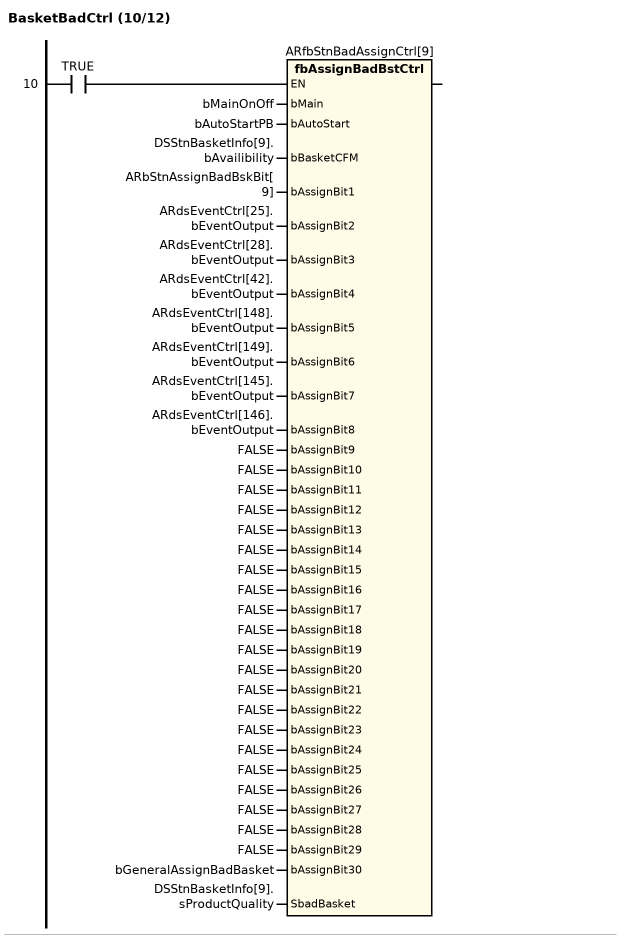
// NETWORK 10
ARfbStnBadAssignCtrl[9](
    bMain := bMainOnOff,
    bAutoStart := bAutoStartPB,
    bBasketCFM := DSStnBasketInfo[9].bAvailibility,
    bAssignBit1 := ARbStnAssignBadBskBit[9],
    bAssignBit2 := ARdsEventCtrl[25].bEventOutput,
    bAssignBit3 := ARdsEventCtrl[28].bEventOutput,
    bAssignBit4 := ARdsEventCtrl[42].bEventOutput,
    bAssignBit5 := ARdsEventCtrl[148].bEventOutput,
    bAssignBit6 := ARdsEventCtrl[149].bEventOutput,
    bAssignBit7 := ARdsEventCtrl[145].bEventOutput,
    bAssignBit8 := ARdsEventCtrl[146].bEventOutput,
    bAssignBit9 := FALSE,
    bAssignBit10 := FALSE,
    bAssignBit11 := FALSE,
    bAssignBit12 := FALSE,
    bAssignBit13 := FALSE,
    bAssignBit14 := FALSE,
    bAssignBit15 := FALSE,
    bAssignBit16 := FALSE,
    bAssignBit17 := FALSE,
    bAssignBit18 := FALSE,
    bAssignBit19 := FALSE,
    bAssignBit20 := FALSE,
    bAssignBit21 := FALSE,
    bAssignBit22 := FALSE,
    bAssignBit23 := FALSE,
    bAssignBit24 := FALSE,
    bAssignBit25 := FALSE,
    bAssignBit26 := FALSE,
    bAssignBit27 := FALSE,
    bAssignBit28 := FALSE,
    bAssignBit29 := FALSE,
    bAssignBit30 := bGeneralAssignBadBasket,
    SbadBasket := DSStnBasketInfo[9].sProductQuality); // fbAssignBadBstCtrl

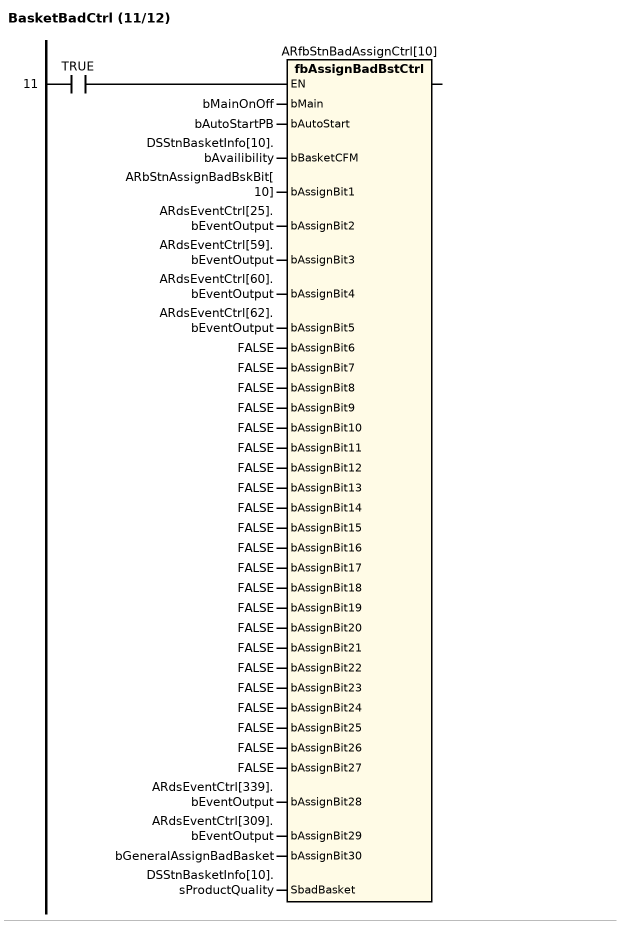
// NETWORK 11
ARfbStnBadAssignCtrl[10](
    bMain := bMainOnOff,
    bAutoStart := bAutoStartPB,
    bBasketCFM := DSStnBasketInfo[10].bAvailibility,
    bAssignBit1 := ARbStnAssignBadBskBit[10],
    bAssignBit2 := ARdsEventCtrl[25].bEventOutput,
    bAssignBit3 := ARdsEventCtrl[59].bEventOutput,
    bAssignBit4 := ARdsEventCtrl[60].bEventOutput,
    bAssignBit5 := ARdsEventCtrl[62].bEventOutput,
    bAssignBit6 := FALSE,
    bAssignBit7 := FALSE,
    bAssignBit8 := FALSE,
    bAssignBit9 := FALSE,
    bAssignBit10 := FALSE,
    bAssignBit11 := FALSE,
    bAssignBit12 := FALSE,
    bAssignBit13 := FALSE,
    bAssignBit14 := FALSE,
    bAssignBit15 := FALSE,
    bAssignBit16 := FALSE,
    bAssignBit17 := FALSE,
    bAssignBit18 := FALSE,
    bAssignBit19 := FALSE,
    bAssignBit20 := FALSE,
    bAssignBit21 := FALSE,
    bAssignBit22 := FALSE,
    bAssignBit23 := FALSE,
    bAssignBit24 := FALSE,
    bAssignBit25 := FALSE,
    bAssignBit26 := FALSE,
    bAssignBit27 := FALSE,
    bAssignBit28 := ARdsEventCtrl[339].bEventOutput,
    bAssignBit29 := ARdsEventCtrl[309].bEventOutput,
    bAssignBit30 := bGeneralAssignBadBasket,
    SbadBasket := DSStnBasketInfo[10].sProductQuality); // fbAssignBadBstCtrl

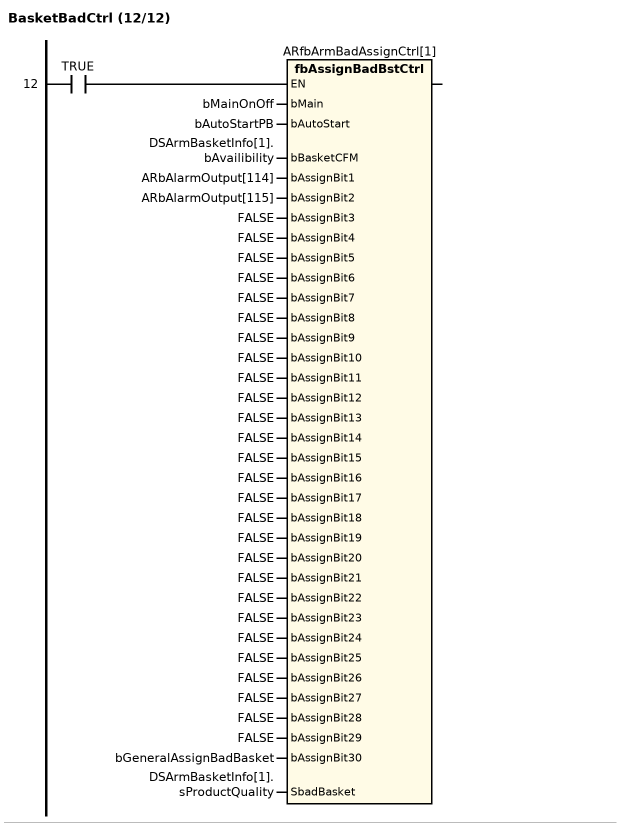
// NETWORK 12
ARfbArmBadAssignCtrl[1](
    bMain := bMainOnOff,
    bAutoStart := bAutoStartPB,
    bBasketCFM := DSArmBasketInfo[1].bAvailibility,
    bAssignBit1 := ARbAlarmOutput[114],
    bAssignBit2 := ARbAlarmOutput[115],
    bAssignBit3 := FALSE,
    bAssignBit4 := FALSE,
    bAssignBit5 := FALSE,
    bAssignBit6 := FALSE,
    bAssignBit7 := FALSE,
    bAssignBit8 := FALSE,
    bAssignBit9 := FALSE,
    bAssignBit10 := FALSE,
    bAssignBit11 := FALSE,
    bAssignBit12 := FALSE,
    bAssignBit13 := FALSE,
    bAssignBit14 := FALSE,
    bAssignBit15 := FALSE,
    bAssignBit16 := FALSE,
    bAssignBit17 := FALSE,
    bAssignBit18 := FALSE,
    bAssignBit19 := FALSE,
    bAssignBit20 := FALSE,
    bAssignBit21 := FALSE,
    bAssignBit22 := FALSE,
    bAssignBit23 := FALSE,
    bAssignBit24 := FALSE,
    bAssignBit25 := FALSE,
    bAssignBit26 := FALSE,
    bAssignBit27 := FALSE,
    bAssignBit28 := FALSE,
    bAssignBit29 := FALSE,
    bAssignBit30 := bGeneralAssignBadBasket,
    SbadBasket := DSArmBasketInfo[1].sProductQuality); // fbAssignBadBstCtrl

END_PROGRAM

// ---- FBs/B_JKS_CustomFB/fbGeneralfbFolder/fbAssignBadBstCtrl.TcPOU
FUNCTION_BLOCK fbAssignBadBstCtrl
VAR_INPUT

	bMain			: BOOL;
	bAutoStart		: BOOL;
	bBasketCFM		: BOOL;

	bAssignBit1		: BOOL;
	bAssignBit2		: BOOL;
	bAssignBit3		: BOOL;
	bAssignBit4		: BOOL;
	bAssignBit5		: BOOL;
	bAssignBit6		: BOOL;
	bAssignBit7		: BOOL;
	bAssignBit8		: BOOL;
	bAssignBit9		: BOOL;
	bAssignBit10		: BOOL;
	bAssignBit11		: BOOL;
	bAssignBit12		: BOOL;
	bAssignBit13		: BOOL;
	bAssignBit14		: BOOL;
	bAssignBit15		: BOOL;
	bAssignBit16		: BOOL;
	bAssignBit17		: BOOL;
	bAssignBit18		: BOOL;
	bAssignBit19		: BOOL;
	bAssignBit20		: BOOL;
	bAssignBit21		: BOOL;
	bAssignBit22		: BOOL;
	bAssignBit23		: BOOL;
	bAssignBit24		: BOOL;
	bAssignBit25		: BOOL;
	bAssignBit26		: BOOL;
	bAssignBit27		: BOOL;
	bAssignBit28		: BOOL;
	bAssignBit29		: BOOL;
	bAssignBit30		: BOOL;

END_VAR
VAR_IN_OUT

	SbadBasket		: STRING(50);

END_VAR
VAR
	TRIG1: R_TRIG;
END_VAR
VAR // added by the converter: edge detectors and wires of the graphical bodies
    _w1 : ANY;
END_VAR

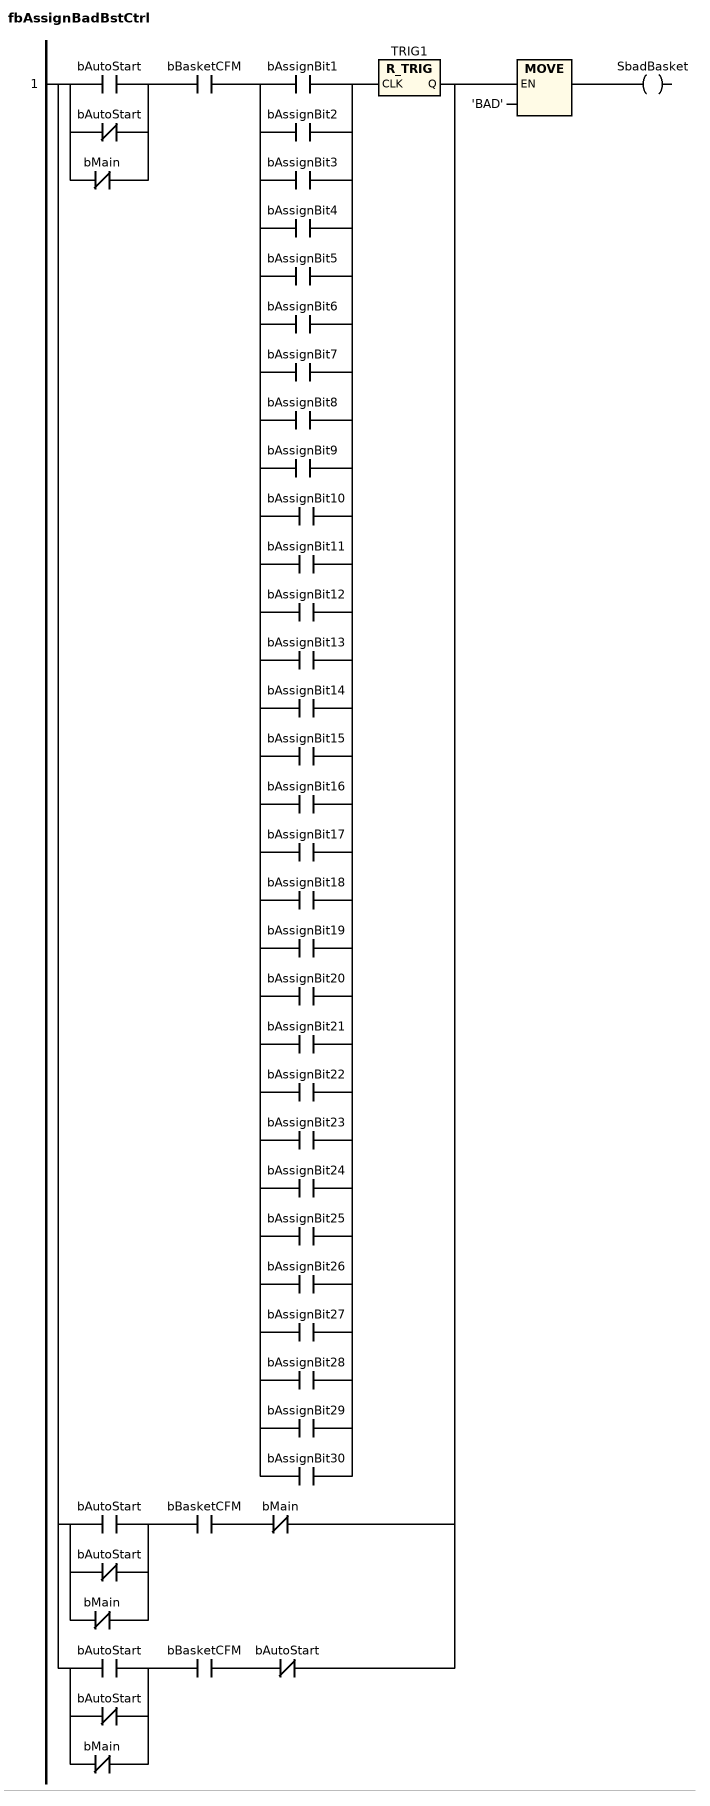
// NETWORK 1
TRIG1(CLK := ((bAutoStart OR NOT bAutoStart OR NOT bMain) AND bBasketCFM) AND (bAssignBit1 OR bAssignBit2 OR bAssignBit3 OR bAssignBit4 OR bAssignBit5 OR bAssignBit6 OR bAssignBit7 OR bAssignBit8 OR bAssignBit9 OR bAssignBit10 OR bAssignBit11 OR bAssignBit12 OR bAssignBit13 OR bAssignBit14 OR bAssignBit15 OR bAssignBit16 OR bAssignBit17 OR bAssignBit18 OR bAssignBit19 OR bAssignBit20 OR bAssignBit21 OR bAssignBit22 OR bAssignBit23 OR bAssignBit24 OR bAssignBit25 OR bAssignBit26 OR bAssignBit27 OR bAssignBit28 OR bAssignBit29 OR bAssignBit30)); // R_TRIG
IF TRIG1.Q OR ((bAutoStart OR NOT bAutoStart OR NOT bMain) AND bBasketCFM) AND NOT bMain OR ((bAutoStart OR NOT bAutoStart OR NOT bMain) AND bBasketCFM) AND NOT bAutoStart THEN
    _w1 := 'BAD';
END_IF
SbadBasket := _w1;

END_FUNCTION_BLOCK

// ---- POUs/MainProgram/BasketMemory_RecipeCtrl/BasketMemoryCtrl.TcPOU
PROGRAM BasketMemoryCtrl
VAR

	NIL: BOOL;

END_VAR

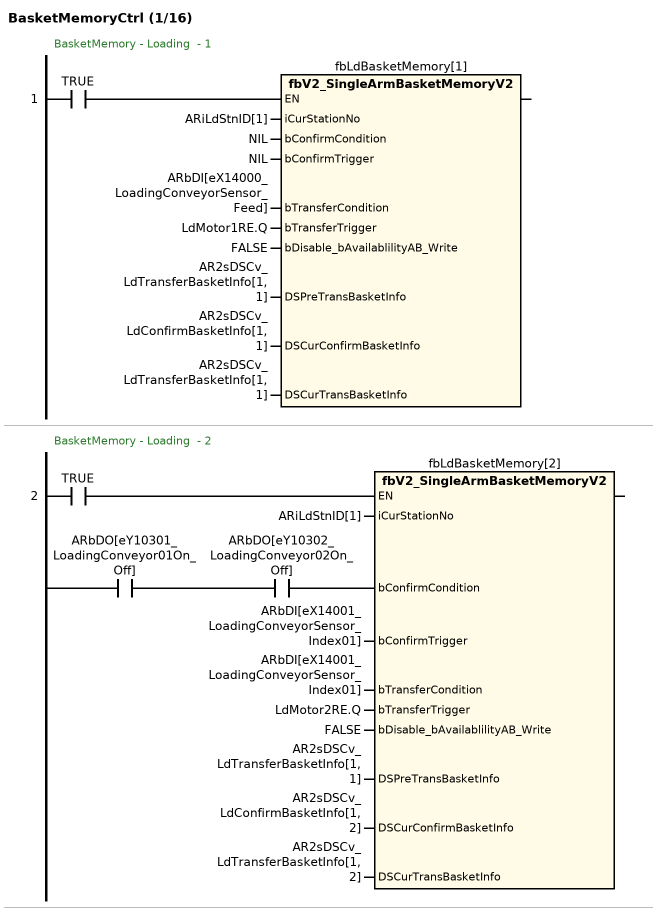
// NETWORK 1
// BasketMemory - Loading  - 1
fbLdBasketMemory[1](
    iCurStationNo := ARiLdStnID[1],
    bConfirmCondition := NIL,
    bConfirmTrigger := NIL,
    bTransferCondition := ARbDI[eX14000_LoadingConveyorSensor_Feed],
    bTransferTrigger := LdMotor1RE.Q,
    bDisable_bAvailablilityAB_Write := FALSE,
    DSPreTransBasketInfo := AR2sDSCv_LdTransferBasketInfo[1,1],
    DSCurConfirmBasketInfo := AR2sDSCv_LdConfirmBasketInfo[1,1],
    DSCurTransBasketInfo := AR2sDSCv_LdTransferBasketInfo[1,1]); // fbV2_SingleArmBasketMemoryV2

// NETWORK 2
// BasketMemory - Loading  - 2
fbLdBasketMemory[2](
    iCurStationNo := ARiLdStnID[1],
    bConfirmCondition := ARbDO[eY10301_LoadingConveyor01On_Off] AND ARbDO[eY10302_LoadingConveyor02On_Off],
    bConfirmTrigger := ARbDI[eX14001_LoadingConveyorSensor_Index01],
    bTransferCondition := ARbDI[eX14001_LoadingConveyorSensor_Index01],
    bTransferTrigger := LdMotor2RE.Q,
    bDisable_bAvailablilityAB_Write := FALSE,
    DSPreTransBasketInfo := AR2sDSCv_LdTransferBasketInfo[1,1],
    DSCurConfirmBasketInfo := AR2sDSCv_LdConfirmBasketInfo[1,2],
    DSCurTransBasketInfo := AR2sDSCv_LdTransferBasketInfo[1,2]); // fbV2_SingleArmBasketMemoryV2

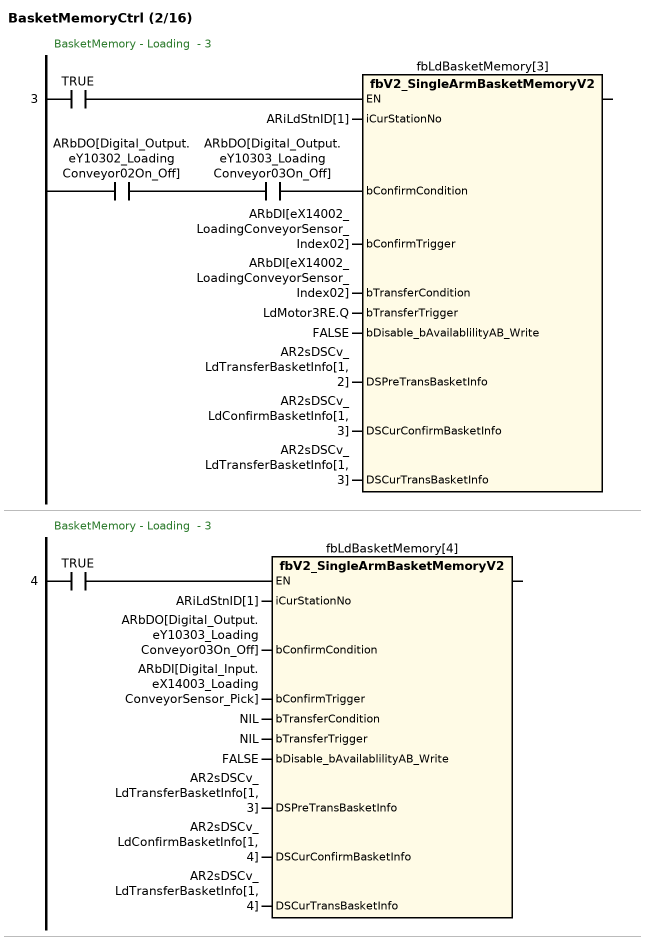
// NETWORK 3
// BasketMemory - Loading  - 3
fbLdBasketMemory[3](
    iCurStationNo := ARiLdStnID[1],
    bConfirmCondition := ARbDO[Digital_Output.eY10302_LoadingConveyor02On_Off] AND ARbDO[Digital_Output.eY10303_LoadingConveyor03On_Off],
    bConfirmTrigger := ARbDI[eX14002_LoadingConveyorSensor_Index02],
    bTransferCondition := ARbDI[eX14002_LoadingConveyorSensor_Index02],
    bTransferTrigger := LdMotor3RE.Q,
    bDisable_bAvailablilityAB_Write := FALSE,
    DSPreTransBasketInfo := AR2sDSCv_LdTransferBasketInfo[1,2],
    DSCurConfirmBasketInfo := AR2sDSCv_LdConfirmBasketInfo[1,3],
    DSCurTransBasketInfo := AR2sDSCv_LdTransferBasketInfo[1,3]); // fbV2_SingleArmBasketMemoryV2

// NETWORK 4
// BasketMemory - Loading  - 3
fbLdBasketMemory[4](
    iCurStationNo := ARiLdStnID[1],
    bConfirmCondition := ARbDO[Digital_Output.eY10303_LoadingConveyor03On_Off],
    bConfirmTrigger := ARbDI[Digital_Input.eX14003_LoadingConveyorSensor_Pick],
    bTransferCondition := NIL,
    bTransferTrigger := NIL,
    bDisable_bAvailablilityAB_Write := FALSE,
    DSPreTransBasketInfo := AR2sDSCv_LdTransferBasketInfo[1,3],
    DSCurConfirmBasketInfo := AR2sDSCv_LdConfirmBasketInfo[1,4],
    DSCurTransBasketInfo := AR2sDSCv_LdTransferBasketInfo[1,4]); // fbV2_SingleArmBasketMemoryV2

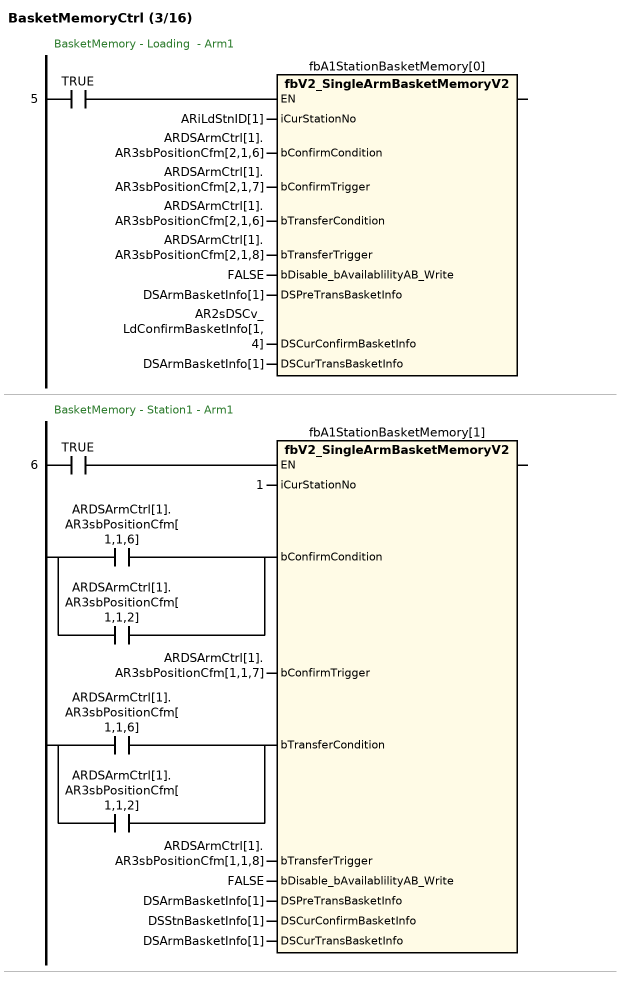
// NETWORK 5
// BasketMemory - Loading  - Arm1
fbA1StationBasketMemory[0](
    iCurStationNo := ARiLdStnID[1],
    bConfirmCondition := ARDSArmCtrl[1].AR3sbPositionCfm[2,1,6],
    bConfirmTrigger := ARDSArmCtrl[1].AR3sbPositionCfm[2,1,7],
    bTransferCondition := ARDSArmCtrl[1].AR3sbPositionCfm[2,1,6],
    bTransferTrigger := ARDSArmCtrl[1].AR3sbPositionCfm[2,1,8],
    bDisable_bAvailablilityAB_Write := FALSE,
    DSPreTransBasketInfo := DSArmBasketInfo[1],
    DSCurConfirmBasketInfo := AR2sDSCv_LdConfirmBasketInfo[1,4],
    DSCurTransBasketInfo := DSArmBasketInfo[1]); // fbV2_SingleArmBasketMemoryV2

// NETWORK 6
// BasketMemory - Station1 - Arm1
fbA1StationBasketMemory[1](
    iCurStationNo := 1,
    bConfirmCondition := ARDSArmCtrl[1].AR3sbPositionCfm[1,1,6] OR ARDSArmCtrl[1].AR3sbPositionCfm[1,1,2],
    bConfirmTrigger := ARDSArmCtrl[1].AR3sbPositionCfm[1,1,7],
    bTransferCondition := ARDSArmCtrl[1].AR3sbPositionCfm[1,1,6] OR ARDSArmCtrl[1].AR3sbPositionCfm[1,1,2],
    bTransferTrigger := ARDSArmCtrl[1].AR3sbPositionCfm[1,1,8],
    bDisable_bAvailablilityAB_Write := FALSE,
    DSPreTransBasketInfo := DSArmBasketInfo[1],
    DSCurConfirmBasketInfo := DSStnBasketInfo[1],
    DSCurTransBasketInfo := DSArmBasketInfo[1]); // fbV2_SingleArmBasketMemoryV2

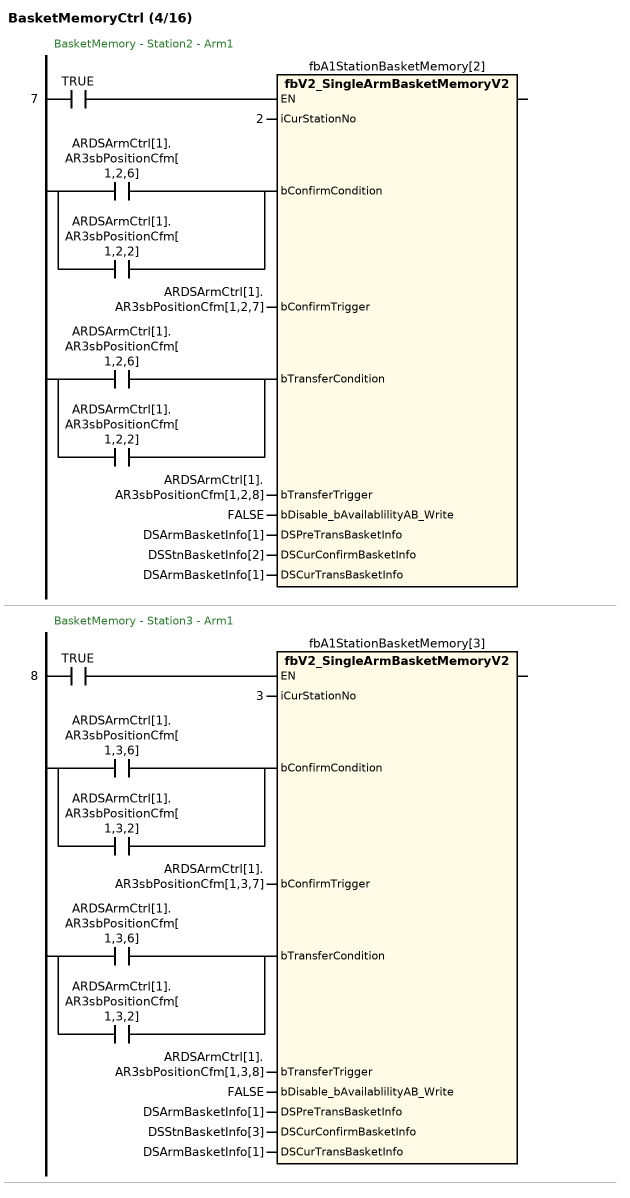
// NETWORK 7
// BasketMemory - Station2 - Arm1
fbA1StationBasketMemory[2](
    iCurStationNo := 2,
    bConfirmCondition := ARDSArmCtrl[1].AR3sbPositionCfm[1,2,6] OR ARDSArmCtrl[1].AR3sbPositionCfm[1,2,2],
    bConfirmTrigger := ARDSArmCtrl[1].AR3sbPositionCfm[1,2,7],
    bTransferCondition := ARDSArmCtrl[1].AR3sbPositionCfm[1,2,6] OR ARDSArmCtrl[1].AR3sbPositionCfm[1,2,2],
    bTransferTrigger := ARDSArmCtrl[1].AR3sbPositionCfm[1,2,8],
    bDisable_bAvailablilityAB_Write := FALSE,
    DSPreTransBasketInfo := DSArmBasketInfo[1],
    DSCurConfirmBasketInfo := DSStnBasketInfo[2],
    DSCurTransBasketInfo := DSArmBasketInfo[1]); // fbV2_SingleArmBasketMemoryV2

// NETWORK 8
// BasketMemory - Station3 - Arm1
fbA1StationBasketMemory[3](
    iCurStationNo := 3,
    bConfirmCondition := ARDSArmCtrl[1].AR3sbPositionCfm[1,3,6] OR ARDSArmCtrl[1].AR3sbPositionCfm[1,3,2],
    bConfirmTrigger := ARDSArmCtrl[1].AR3sbPositionCfm[1,3,7],
    bTransferCondition := ARDSArmCtrl[1].AR3sbPositionCfm[1,3,6] OR ARDSArmCtrl[1].AR3sbPositionCfm[1,3,2],
    bTransferTrigger := ARDSArmCtrl[1].AR3sbPositionCfm[1,3,8],
    bDisable_bAvailablilityAB_Write := FALSE,
    DSPreTransBasketInfo := DSArmBasketInfo[1],
    DSCurConfirmBasketInfo := DSStnBasketInfo[3],
    DSCurTransBasketInfo := DSArmBasketInfo[1]); // fbV2_SingleArmBasketMemoryV2

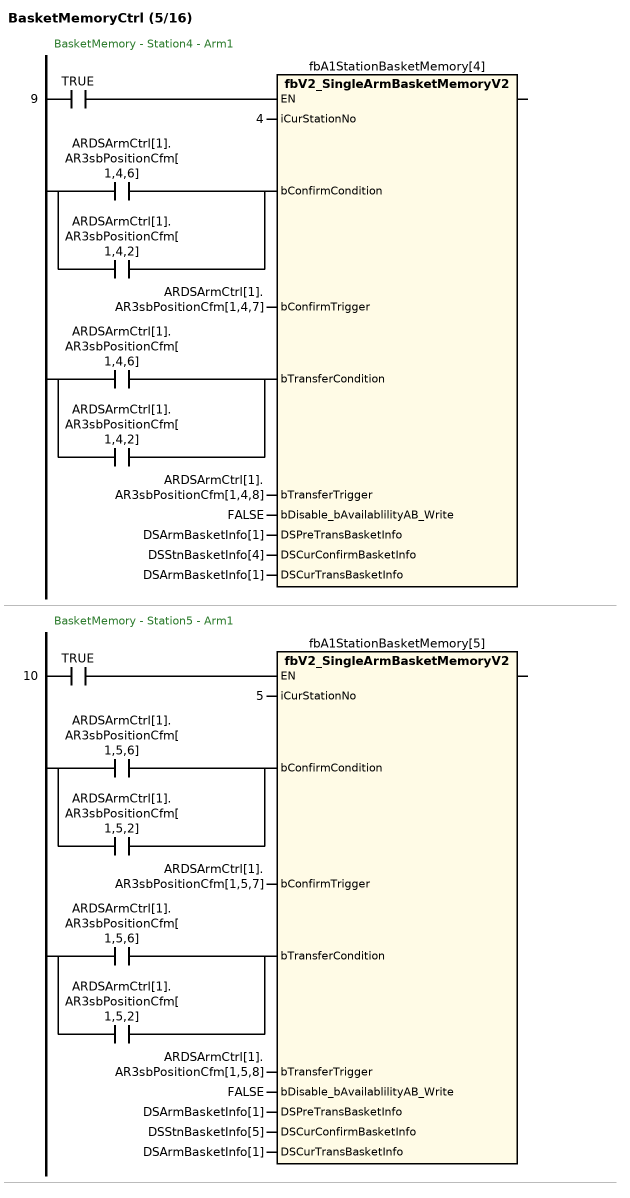
// NETWORK 9
// BasketMemory - Station4 - Arm1
fbA1StationBasketMemory[4](
    iCurStationNo := 4,
    bConfirmCondition := ARDSArmCtrl[1].AR3sbPositionCfm[1,4,6] OR ARDSArmCtrl[1].AR3sbPositionCfm[1,4,2],
    bConfirmTrigger := ARDSArmCtrl[1].AR3sbPositionCfm[1,4,7],
    bTransferCondition := ARDSArmCtrl[1].AR3sbPositionCfm[1,4,6] OR ARDSArmCtrl[1].AR3sbPositionCfm[1,4,2],
    bTransferTrigger := ARDSArmCtrl[1].AR3sbPositionCfm[1,4,8],
    bDisable_bAvailablilityAB_Write := FALSE,
    DSPreTransBasketInfo := DSArmBasketInfo[1],
    DSCurConfirmBasketInfo := DSStnBasketInfo[4],
    DSCurTransBasketInfo := DSArmBasketInfo[1]); // fbV2_SingleArmBasketMemoryV2

// NETWORK 10
// BasketMemory - Station5 - Arm1
fbA1StationBasketMemory[5](
    iCurStationNo := 5,
    bConfirmCondition := ARDSArmCtrl[1].AR3sbPositionCfm[1,5,6] OR ARDSArmCtrl[1].AR3sbPositionCfm[1,5,2],
    bConfirmTrigger := ARDSArmCtrl[1].AR3sbPositionCfm[1,5,7],
    bTransferCondition := ARDSArmCtrl[1].AR3sbPositionCfm[1,5,6] OR ARDSArmCtrl[1].AR3sbPositionCfm[1,5,2],
    bTransferTrigger := ARDSArmCtrl[1].AR3sbPositionCfm[1,5,8],
    bDisable_bAvailablilityAB_Write := FALSE,
    DSPreTransBasketInfo := DSArmBasketInfo[1],
    DSCurConfirmBasketInfo := DSStnBasketInfo[5],
    DSCurTransBasketInfo := DSArmBasketInfo[1]); // fbV2_SingleArmBasketMemoryV2

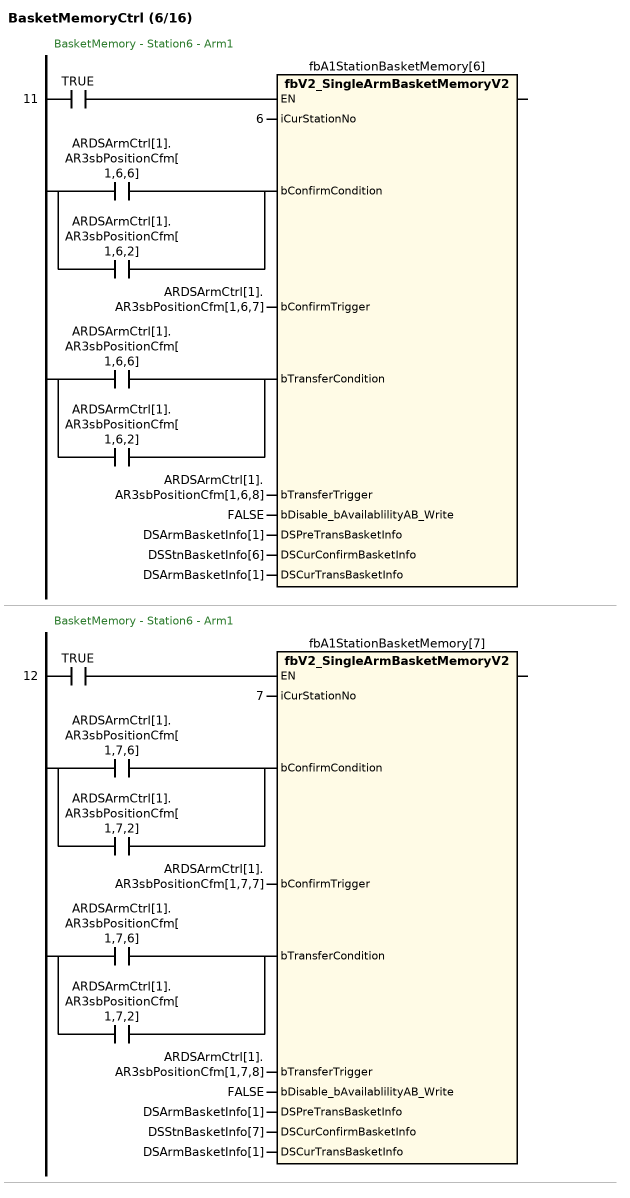
// NETWORK 11
// BasketMemory - Station6 - Arm1
fbA1StationBasketMemory[6](
    iCurStationNo := 6,
    bConfirmCondition := ARDSArmCtrl[1].AR3sbPositionCfm[1,6,6] OR ARDSArmCtrl[1].AR3sbPositionCfm[1,6,2],
    bConfirmTrigger := ARDSArmCtrl[1].AR3sbPositionCfm[1,6,7],
    bTransferCondition := ARDSArmCtrl[1].AR3sbPositionCfm[1,6,6] OR ARDSArmCtrl[1].AR3sbPositionCfm[1,6,2],
    bTransferTrigger := ARDSArmCtrl[1].AR3sbPositionCfm[1,6,8],
    bDisable_bAvailablilityAB_Write := FALSE,
    DSPreTransBasketInfo := DSArmBasketInfo[1],
    DSCurConfirmBasketInfo := DSStnBasketInfo[6],
    DSCurTransBasketInfo := DSArmBasketInfo[1]); // fbV2_SingleArmBasketMemoryV2

// NETWORK 12
// BasketMemory - Station6 - Arm1
fbA1StationBasketMemory[7](
    iCurStationNo := 7,
    bConfirmCondition := ARDSArmCtrl[1].AR3sbPositionCfm[1,7,6] OR ARDSArmCtrl[1].AR3sbPositionCfm[1,7,2],
    bConfirmTrigger := ARDSArmCtrl[1].AR3sbPositionCfm[1,7,7],
    bTransferCondition := ARDSArmCtrl[1].AR3sbPositionCfm[1,7,6] OR ARDSArmCtrl[1].AR3sbPositionCfm[1,7,2],
    bTransferTrigger := ARDSArmCtrl[1].AR3sbPositionCfm[1,7,8],
    bDisable_bAvailablilityAB_Write := FALSE,
    DSPreTransBasketInfo := DSArmBasketInfo[1],
    DSCurConfirmBasketInfo := DSStnBasketInfo[7],
    DSCurTransBasketInfo := DSArmBasketInfo[1]); // fbV2_SingleArmBasketMemoryV2

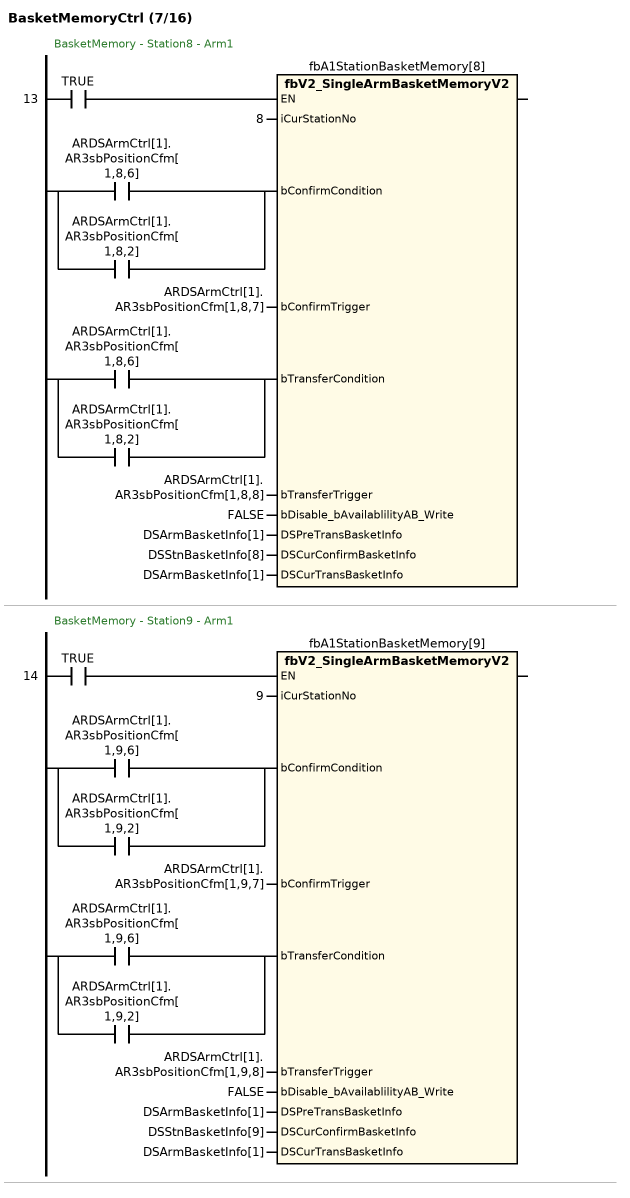
// NETWORK 13
// BasketMemory - Station8 - Arm1
fbA1StationBasketMemory[8](
    iCurStationNo := 8,
    bConfirmCondition := ARDSArmCtrl[1].AR3sbPositionCfm[1,8,6] OR ARDSArmCtrl[1].AR3sbPositionCfm[1,8,2],
    bConfirmTrigger := ARDSArmCtrl[1].AR3sbPositionCfm[1,8,7],
    bTransferCondition := ARDSArmCtrl[1].AR3sbPositionCfm[1,8,6] OR ARDSArmCtrl[1].AR3sbPositionCfm[1,8,2],
    bTransferTrigger := ARDSArmCtrl[1].AR3sbPositionCfm[1,8,8],
    bDisable_bAvailablilityAB_Write := FALSE,
    DSPreTransBasketInfo := DSArmBasketInfo[1],
    DSCurConfirmBasketInfo := DSStnBasketInfo[8],
    DSCurTransBasketInfo := DSArmBasketInfo[1]); // fbV2_SingleArmBasketMemoryV2

// NETWORK 14
// BasketMemory - Station9 - Arm1
fbA1StationBasketMemory[9](
    iCurStationNo := 9,
    bConfirmCondition := ARDSArmCtrl[1].AR3sbPositionCfm[1,9,6] OR ARDSArmCtrl[1].AR3sbPositionCfm[1,9,2],
    bConfirmTrigger := ARDSArmCtrl[1].AR3sbPositionCfm[1,9,7],
    bTransferCondition := ARDSArmCtrl[1].AR3sbPositionCfm[1,9,6] OR ARDSArmCtrl[1].AR3sbPositionCfm[1,9,2],
    bTransferTrigger := ARDSArmCtrl[1].AR3sbPositionCfm[1,9,8],
    bDisable_bAvailablilityAB_Write := FALSE,
    DSPreTransBasketInfo := DSArmBasketInfo[1],
    DSCurConfirmBasketInfo := DSStnBasketInfo[9],
    DSCurTransBasketInfo := DSArmBasketInfo[1]); // fbV2_SingleArmBasketMemoryV2

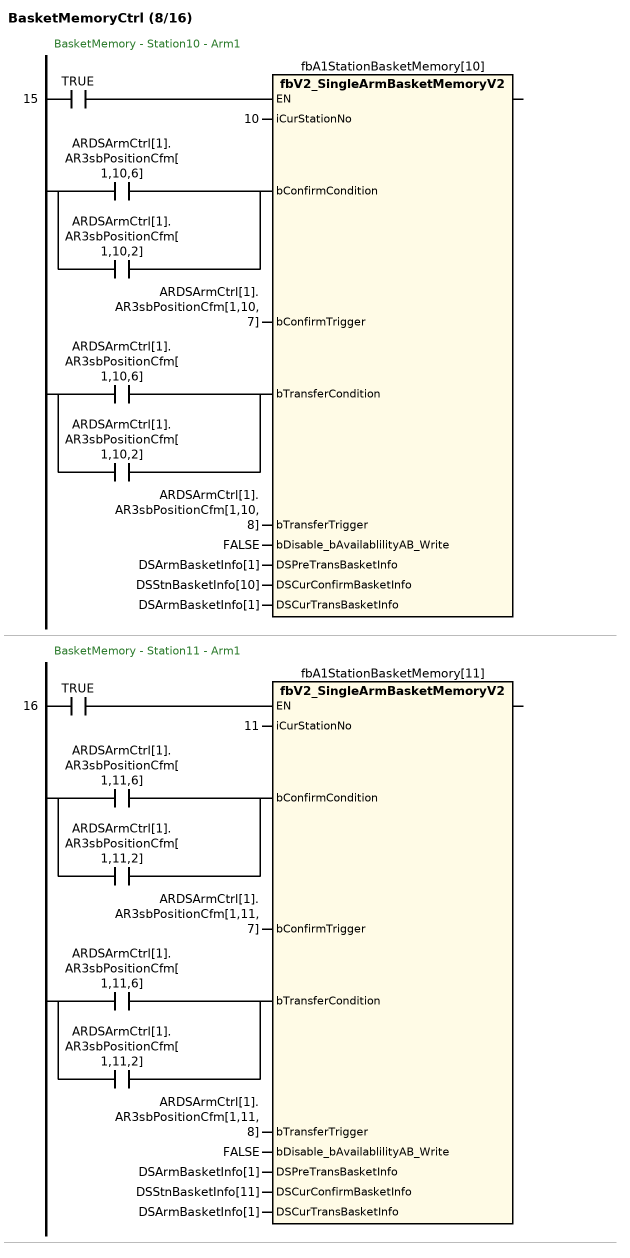
// NETWORK 15
// BasketMemory - Station10 - Arm1
fbA1StationBasketMemory[10](
    iCurStationNo := 10,
    bConfirmCondition := ARDSArmCtrl[1].AR3sbPositionCfm[1,10,6] OR ARDSArmCtrl[1].AR3sbPositionCfm[1,10,2],
    bConfirmTrigger := ARDSArmCtrl[1].AR3sbPositionCfm[1,10,7],
    bTransferCondition := ARDSArmCtrl[1].AR3sbPositionCfm[1,10,6] OR ARDSArmCtrl[1].AR3sbPositionCfm[1,10,2],
    bTransferTrigger := ARDSArmCtrl[1].AR3sbPositionCfm[1,10,8],
    bDisable_bAvailablilityAB_Write := FALSE,
    DSPreTransBasketInfo := DSArmBasketInfo[1],
    DSCurConfirmBasketInfo := DSStnBasketInfo[10],
    DSCurTransBasketInfo := DSArmBasketInfo[1]); // fbV2_SingleArmBasketMemoryV2

// NETWORK 16
// BasketMemory - Station11 - Arm1
fbA1StationBasketMemory[11](
    iCurStationNo := 11,
    bConfirmCondition := ARDSArmCtrl[1].AR3sbPositionCfm[1,11,6] OR ARDSArmCtrl[1].AR3sbPositionCfm[1,11,2],
    bConfirmTrigger := ARDSArmCtrl[1].AR3sbPositionCfm[1,11,7],
    bTransferCondition := ARDSArmCtrl[1].AR3sbPositionCfm[1,11,6] OR ARDSArmCtrl[1].AR3sbPositionCfm[1,11,2],
    bTransferTrigger := ARDSArmCtrl[1].AR3sbPositionCfm[1,11,8],
    bDisable_bAvailablilityAB_Write := FALSE,
    DSPreTransBasketInfo := DSArmBasketInfo[1],
    DSCurConfirmBasketInfo := DSStnBasketInfo[11],
    DSCurTransBasketInfo := DSArmBasketInfo[1]); // fbV2_SingleArmBasketMemoryV2

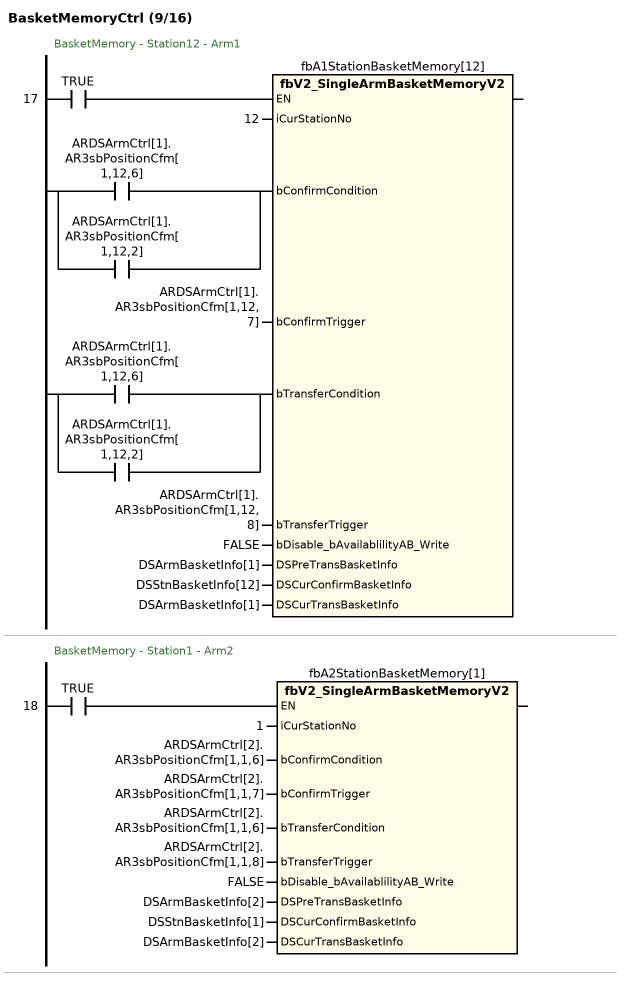
// NETWORK 17
// BasketMemory - Station12 - Arm1
fbA1StationBasketMemory[12](
    iCurStationNo := 12,
    bConfirmCondition := ARDSArmCtrl[1].AR3sbPositionCfm[1,12,6] OR ARDSArmCtrl[1].AR3sbPositionCfm[1,12,2],
    bConfirmTrigger := ARDSArmCtrl[1].AR3sbPositionCfm[1,12,7],
    bTransferCondition := ARDSArmCtrl[1].AR3sbPositionCfm[1,12,6] OR ARDSArmCtrl[1].AR3sbPositionCfm[1,12,2],
    bTransferTrigger := ARDSArmCtrl[1].AR3sbPositionCfm[1,12,8],
    bDisable_bAvailablilityAB_Write := FALSE,
    DSPreTransBasketInfo := DSArmBasketInfo[1],
    DSCurConfirmBasketInfo := DSStnBasketInfo[12],
    DSCurTransBasketInfo := DSArmBasketInfo[1]); // fbV2_SingleArmBasketMemoryV2

// NETWORK 18
// BasketMemory - Station1 - Arm2
fbA2StationBasketMemory[1](
    iCurStationNo := 1,
    bConfirmCondition := ARDSArmCtrl[2].AR3sbPositionCfm[1,1,6],
    bConfirmTrigger := ARDSArmCtrl[2].AR3sbPositionCfm[1,1,7],
    bTransferCondition := ARDSArmCtrl[2].AR3sbPositionCfm[1,1,6],
    bTransferTrigger := ARDSArmCtrl[2].AR3sbPositionCfm[1,1,8],
    bDisable_bAvailablilityAB_Write := FALSE,
    DSPreTransBasketInfo := DSArmBasketInfo[2],
    DSCurConfirmBasketInfo := DSStnBasketInfo[1],
    DSCurTransBasketInfo := DSArmBasketInfo[2]); // fbV2_SingleArmBasketMemoryV2

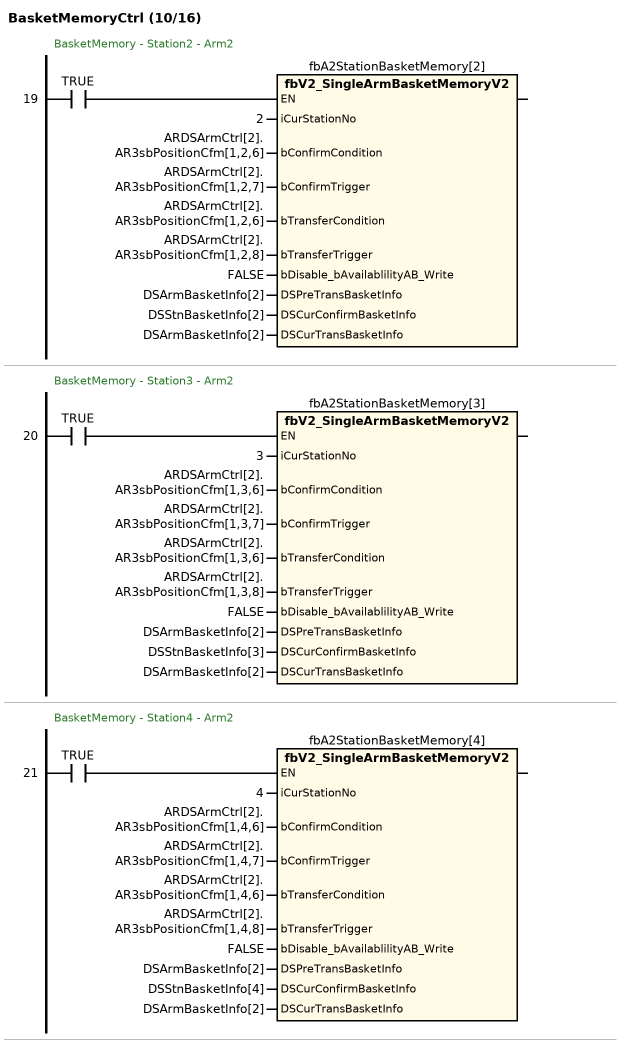
// NETWORK 19
// BasketMemory - Station2 - Arm2
fbA2StationBasketMemory[2](
    iCurStationNo := 2,
    bConfirmCondition := ARDSArmCtrl[2].AR3sbPositionCfm[1,2,6],
    bConfirmTrigger := ARDSArmCtrl[2].AR3sbPositionCfm[1,2,7],
    bTransferCondition := ARDSArmCtrl[2].AR3sbPositionCfm[1,2,6],
    bTransferTrigger := ARDSArmCtrl[2].AR3sbPositionCfm[1,2,8],
    bDisable_bAvailablilityAB_Write := FALSE,
    DSPreTransBasketInfo := DSArmBasketInfo[2],
    DSCurConfirmBasketInfo := DSStnBasketInfo[2],
    DSCurTransBasketInfo := DSArmBasketInfo[2]); // fbV2_SingleArmBasketMemoryV2

// NETWORK 20
// BasketMemory - Station3 - Arm2
fbA2StationBasketMemory[3](
    iCurStationNo := 3,
    bConfirmCondition := ARDSArmCtrl[2].AR3sbPositionCfm[1,3,6],
    bConfirmTrigger := ARDSArmCtrl[2].AR3sbPositionCfm[1,3,7],
    bTransferCondition := ARDSArmCtrl[2].AR3sbPositionCfm[1,3,6],
    bTransferTrigger := ARDSArmCtrl[2].AR3sbPositionCfm[1,3,8],
    bDisable_bAvailablilityAB_Write := FALSE,
    DSPreTransBasketInfo := DSArmBasketInfo[2],
    DSCurConfirmBasketInfo := DSStnBasketInfo[3],
    DSCurTransBasketInfo := DSArmBasketInfo[2]); // fbV2_SingleArmBasketMemoryV2

// NETWORK 21
// BasketMemory - Station4 - Arm2
fbA2StationBasketMemory[4](
    iCurStationNo := 4,
    bConfirmCondition := ARDSArmCtrl[2].AR3sbPositionCfm[1,4,6],
    bConfirmTrigger := ARDSArmCtrl[2].AR3sbPositionCfm[1,4,7],
    bTransferCondition := ARDSArmCtrl[2].AR3sbPositionCfm[1,4,6],
    bTransferTrigger := ARDSArmCtrl[2].AR3sbPositionCfm[1,4,8],
    bDisable_bAvailablilityAB_Write := FALSE,
    DSPreTransBasketInfo := DSArmBasketInfo[2],
    DSCurConfirmBasketInfo := DSStnBasketInfo[4],
    DSCurTransBasketInfo := DSArmBasketInfo[2]); // fbV2_SingleArmBasketMemoryV2

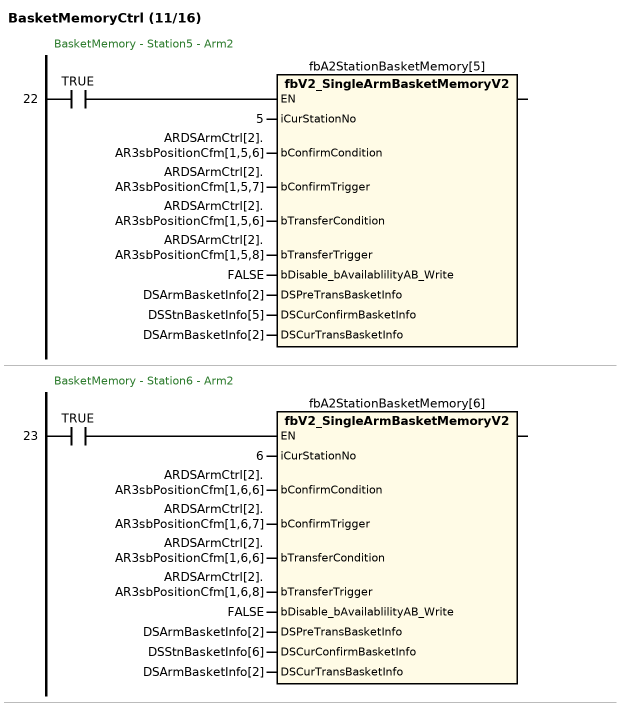
// NETWORK 22
// BasketMemory - Station5 - Arm2
fbA2StationBasketMemory[5](
    iCurStationNo := 5,
    bConfirmCondition := ARDSArmCtrl[2].AR3sbPositionCfm[1,5,6],
    bConfirmTrigger := ARDSArmCtrl[2].AR3sbPositionCfm[1,5,7],
    bTransferCondition := ARDSArmCtrl[2].AR3sbPositionCfm[1,5,6],
    bTransferTrigger := ARDSArmCtrl[2].AR3sbPositionCfm[1,5,8],
    bDisable_bAvailablilityAB_Write := FALSE,
    DSPreTransBasketInfo := DSArmBasketInfo[2],
    DSCurConfirmBasketInfo := DSStnBasketInfo[5],
    DSCurTransBasketInfo := DSArmBasketInfo[2]); // fbV2_SingleArmBasketMemoryV2

// NETWORK 23
// BasketMemory - Station6 - Arm2
fbA2StationBasketMemory[6](
    iCurStationNo := 6,
    bConfirmCondition := ARDSArmCtrl[2].AR3sbPositionCfm[1,6,6],
    bConfirmTrigger := ARDSArmCtrl[2].AR3sbPositionCfm[1,6,7],
    bTransferCondition := ARDSArmCtrl[2].AR3sbPositionCfm[1,6,6],
    bTransferTrigger := ARDSArmCtrl[2].AR3sbPositionCfm[1,6,8],
    bDisable_bAvailablilityAB_Write := FALSE,
    DSPreTransBasketInfo := DSArmBasketInfo[2],
    DSCurConfirmBasketInfo := DSStnBasketInfo[6],
    DSCurTransBasketInfo := DSArmBasketInfo[2]); // fbV2_SingleArmBasketMemoryV2

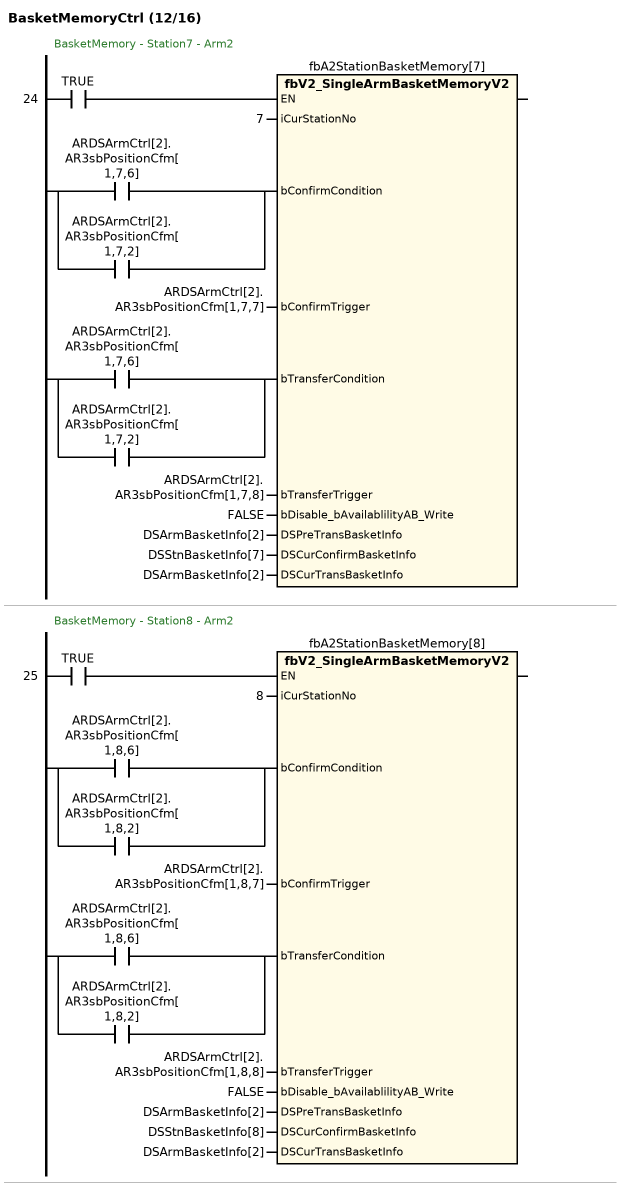
// NETWORK 24
// BasketMemory - Station7 - Arm2
fbA2StationBasketMemory[7](
    iCurStationNo := 7,
    bConfirmCondition := ARDSArmCtrl[2].AR3sbPositionCfm[1,7,6] OR ARDSArmCtrl[2].AR3sbPositionCfm[1,7,2],
    bConfirmTrigger := ARDSArmCtrl[2].AR3sbPositionCfm[1,7,7],
    bTransferCondition := ARDSArmCtrl[2].AR3sbPositionCfm[1,7,6] OR ARDSArmCtrl[2].AR3sbPositionCfm[1,7,2],
    bTransferTrigger := ARDSArmCtrl[2].AR3sbPositionCfm[1,7,8],
    bDisable_bAvailablilityAB_Write := FALSE,
    DSPreTransBasketInfo := DSArmBasketInfo[2],
    DSCurConfirmBasketInfo := DSStnBasketInfo[7],
    DSCurTransBasketInfo := DSArmBasketInfo[2]); // fbV2_SingleArmBasketMemoryV2

// NETWORK 25
// BasketMemory - Station8 - Arm2
fbA2StationBasketMemory[8](
    iCurStationNo := 8,
    bConfirmCondition := ARDSArmCtrl[2].AR3sbPositionCfm[1,8,6] OR ARDSArmCtrl[2].AR3sbPositionCfm[1,8,2],
    bConfirmTrigger := ARDSArmCtrl[2].AR3sbPositionCfm[1,8,7],
    bTransferCondition := ARDSArmCtrl[2].AR3sbPositionCfm[1,8,6] OR ARDSArmCtrl[2].AR3sbPositionCfm[1,8,2],
    bTransferTrigger := ARDSArmCtrl[2].AR3sbPositionCfm[1,8,8],
    bDisable_bAvailablilityAB_Write := FALSE,
    DSPreTransBasketInfo := DSArmBasketInfo[2],
    DSCurConfirmBasketInfo := DSStnBasketInfo[8],
    DSCurTransBasketInfo := DSArmBasketInfo[2]); // fbV2_SingleArmBasketMemoryV2

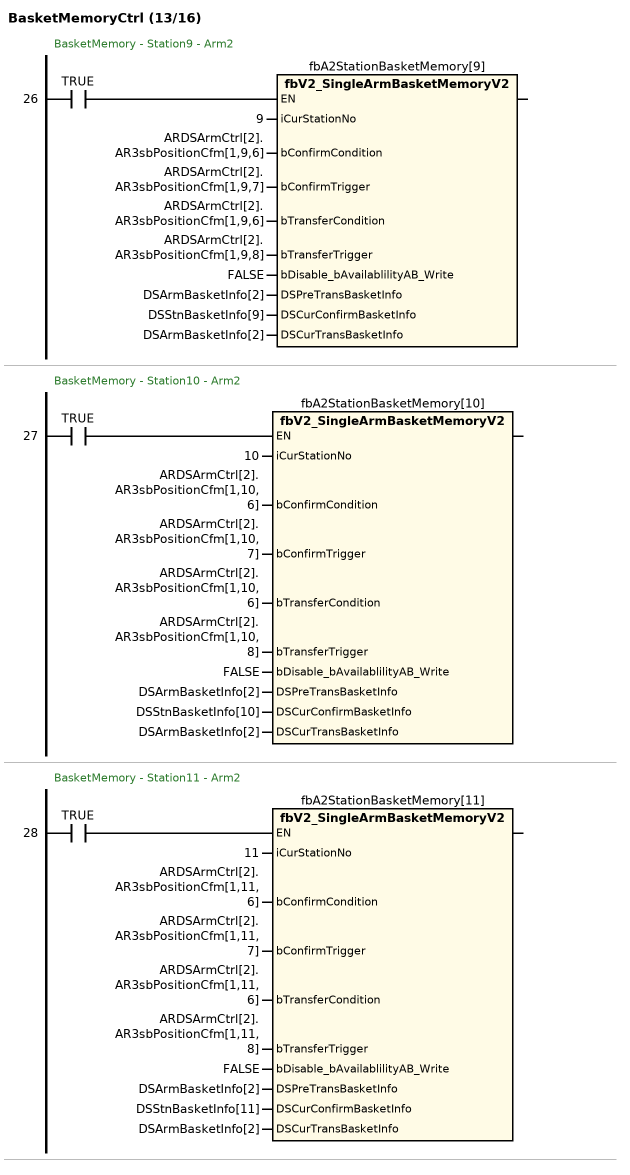
// NETWORK 26
// BasketMemory - Station9 - Arm2
fbA2StationBasketMemory[9](
    iCurStationNo := 9,
    bConfirmCondition := ARDSArmCtrl[2].AR3sbPositionCfm[1,9,6],
    bConfirmTrigger := ARDSArmCtrl[2].AR3sbPositionCfm[1,9,7],
    bTransferCondition := ARDSArmCtrl[2].AR3sbPositionCfm[1,9,6],
    bTransferTrigger := ARDSArmCtrl[2].AR3sbPositionCfm[1,9,8],
    bDisable_bAvailablilityAB_Write := FALSE,
    DSPreTransBasketInfo := DSArmBasketInfo[2],
    DSCurConfirmBasketInfo := DSStnBasketInfo[9],
    DSCurTransBasketInfo := DSArmBasketInfo[2]); // fbV2_SingleArmBasketMemoryV2

// NETWORK 27
// BasketMemory - Station10 - Arm2
fbA2StationBasketMemory[10](
    iCurStationNo := 10,
    bConfirmCondition := ARDSArmCtrl[2].AR3sbPositionCfm[1,10,6],
    bConfirmTrigger := ARDSArmCtrl[2].AR3sbPositionCfm[1,10,7],
    bTransferCondition := ARDSArmCtrl[2].AR3sbPositionCfm[1,10,6],
    bTransferTrigger := ARDSArmCtrl[2].AR3sbPositionCfm[1,10,8],
    bDisable_bAvailablilityAB_Write := FALSE,
    DSPreTransBasketInfo := DSArmBasketInfo[2],
    DSCurConfirmBasketInfo := DSStnBasketInfo[10],
    DSCurTransBasketInfo := DSArmBasketInfo[2]); // fbV2_SingleArmBasketMemoryV2

// NETWORK 28
// BasketMemory - Station11 - Arm2
fbA2StationBasketMemory[11](
    iCurStationNo := 11,
    bConfirmCondition := ARDSArmCtrl[2].AR3sbPositionCfm[1,11,6],
    bConfirmTrigger := ARDSArmCtrl[2].AR3sbPositionCfm[1,11,7],
    bTransferCondition := ARDSArmCtrl[2].AR3sbPositionCfm[1,11,6],
    bTransferTrigger := ARDSArmCtrl[2].AR3sbPositionCfm[1,11,8],
    bDisable_bAvailablilityAB_Write := FALSE,
    DSPreTransBasketInfo := DSArmBasketInfo[2],
    DSCurConfirmBasketInfo := DSStnBasketInfo[11],
    DSCurTransBasketInfo := DSArmBasketInfo[2]); // fbV2_SingleArmBasketMemoryV2

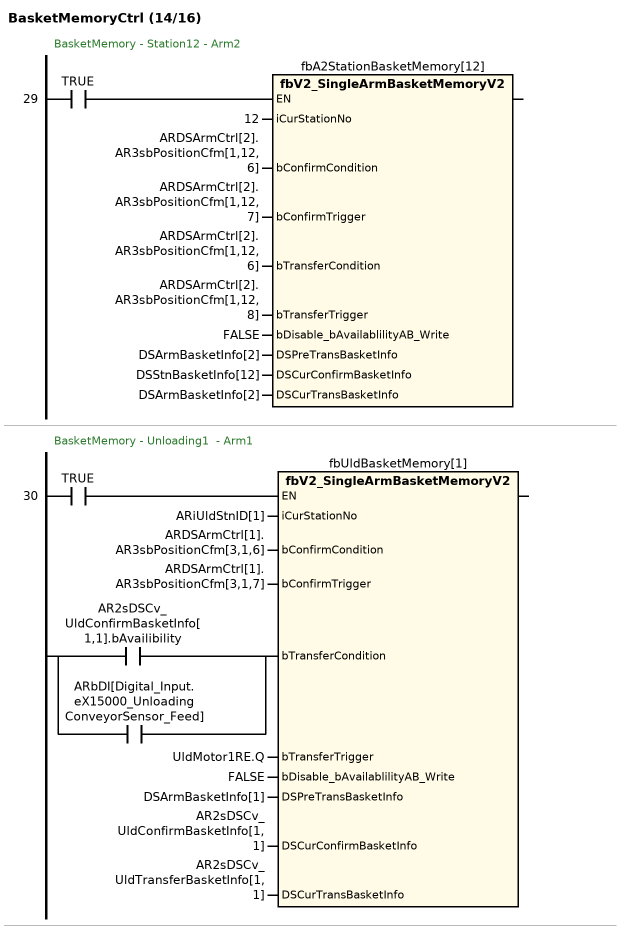
// NETWORK 29
// BasketMemory - Station12 - Arm2
fbA2StationBasketMemory[12](
    iCurStationNo := 12,
    bConfirmCondition := ARDSArmCtrl[2].AR3sbPositionCfm[1,12,6],
    bConfirmTrigger := ARDSArmCtrl[2].AR3sbPositionCfm[1,12,7],
    bTransferCondition := ARDSArmCtrl[2].AR3sbPositionCfm[1,12,6],
    bTransferTrigger := ARDSArmCtrl[2].AR3sbPositionCfm[1,12,8],
    bDisable_bAvailablilityAB_Write := FALSE,
    DSPreTransBasketInfo := DSArmBasketInfo[2],
    DSCurConfirmBasketInfo := DSStnBasketInfo[12],
    DSCurTransBasketInfo := DSArmBasketInfo[2]); // fbV2_SingleArmBasketMemoryV2

// NETWORK 30
// BasketMemory - Unloading1  - Arm1
fbUldBasketMemory[1](
    iCurStationNo := ARiUldStnID[1],
    bConfirmCondition := ARDSArmCtrl[1].AR3sbPositionCfm[3,1,6],
    bConfirmTrigger := ARDSArmCtrl[1].AR3sbPositionCfm[3,1,7],
    bTransferCondition := AR2sDSCv_UldConfirmBasketInfo[1,1].bAvailibility OR ARbDI[Digital_Input.eX15000_UnloadingConveyorSensor_Feed],
    bTransferTrigger := UldMotor1RE.Q,
    bDisable_bAvailablilityAB_Write := FALSE,
    DSPreTransBasketInfo := DSArmBasketInfo[1],
    DSCurConfirmBasketInfo := AR2sDSCv_UldConfirmBasketInfo[1,1],
    DSCurTransBasketInfo := AR2sDSCv_UldTransferBasketInfo[1,1]); // fbV2_SingleArmBasketMemoryV2

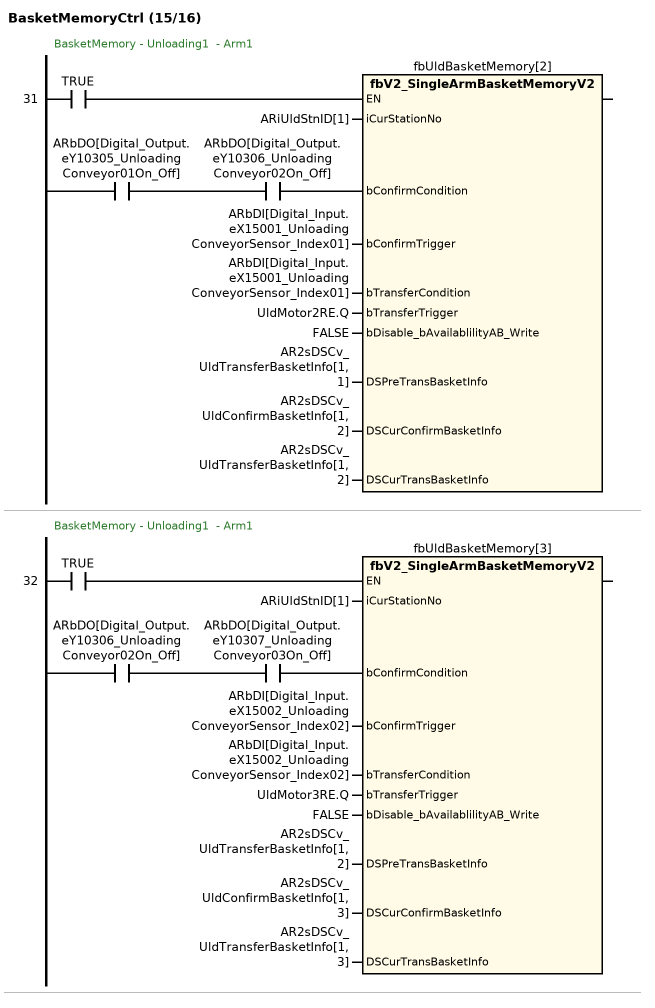
// NETWORK 31
// BasketMemory - Unloading1  - Arm1
fbUldBasketMemory[2](
    iCurStationNo := ARiUldStnID[1],
    bConfirmCondition := ARbDO[Digital_Output.eY10305_UnloadingConveyor01On_Off] AND ARbDO[Digital_Output.eY10306_UnloadingConveyor02On_Off],
    bConfirmTrigger := ARbDI[Digital_Input.eX15001_UnloadingConveyorSensor_Index01],
    bTransferCondition := ARbDI[Digital_Input.eX15001_UnloadingConveyorSensor_Index01],
    bTransferTrigger := UldMotor2RE.Q,
    bDisable_bAvailablilityAB_Write := FALSE,
    DSPreTransBasketInfo := AR2sDSCv_UldTransferBasketInfo[1,1],
    DSCurConfirmBasketInfo := AR2sDSCv_UldConfirmBasketInfo[1,2],
    DSCurTransBasketInfo := AR2sDSCv_UldTransferBasketInfo[1,2]); // fbV2_SingleArmBasketMemoryV2

// NETWORK 32
// BasketMemory - Unloading1  - Arm1
fbUldBasketMemory[3](
    iCurStationNo := ARiUldStnID[1],
    bConfirmCondition := ARbDO[Digital_Output.eY10306_UnloadingConveyor02On_Off] AND ARbDO[Digital_Output.eY10307_UnloadingConveyor03On_Off],
    bConfirmTrigger := ARbDI[Digital_Input.eX15002_UnloadingConveyorSensor_Index02],
    bTransferCondition := ARbDI[Digital_Input.eX15002_UnloadingConveyorSensor_Index02],
    bTransferTrigger := UldMotor3RE.Q,
    bDisable_bAvailablilityAB_Write := FALSE,
    DSPreTransBasketInfo := AR2sDSCv_UldTransferBasketInfo[1,2],
    DSCurConfirmBasketInfo := AR2sDSCv_UldConfirmBasketInfo[1,3],
    DSCurTransBasketInfo := AR2sDSCv_UldTransferBasketInfo[1,3]); // fbV2_SingleArmBasketMemoryV2

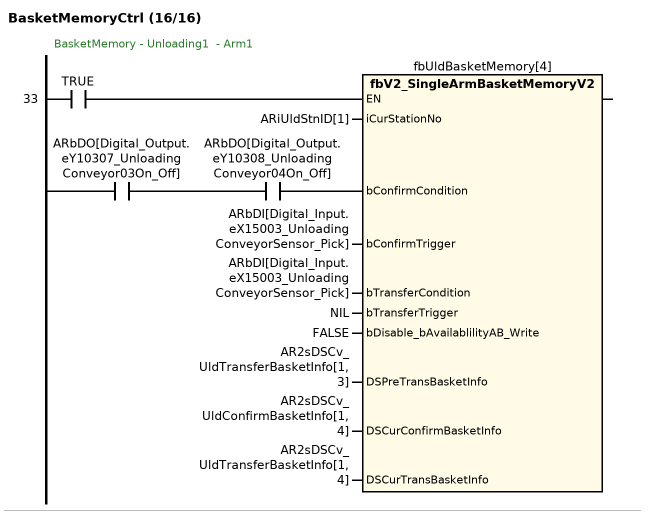
// NETWORK 33
// BasketMemory - Unloading1  - Arm1
fbUldBasketMemory[4](
    iCurStationNo := ARiUldStnID[1],
    bConfirmCondition := ARbDO[Digital_Output.eY10307_UnloadingConveyor03On_Off] AND ARbDO[Digital_Output.eY10308_UnloadingConveyor04On_Off],
    bConfirmTrigger := ARbDI[Digital_Input.eX15003_UnloadingConveyorSensor_Pick],
    bTransferCondition := ARbDI[Digital_Input.eX15003_UnloadingConveyorSensor_Pick],
    bTransferTrigger := NIL,
    bDisable_bAvailablilityAB_Write := FALSE,
    DSPreTransBasketInfo := AR2sDSCv_UldTransferBasketInfo[1,3],
    DSCurConfirmBasketInfo := AR2sDSCv_UldConfirmBasketInfo[1,4],
    DSCurTransBasketInfo := AR2sDSCv_UldTransferBasketInfo[1,4]); // fbV2_SingleArmBasketMemoryV2

END_PROGRAM

// ---- FBs/B_JKS_NewFB_V2/FBP-Memory_Sub/fbV2_SingleArmBasketMemoryV2.TcPOU
FUNCTION_BLOCK fbV2_SingleArmBasketMemoryV2
VAR_INPUT

	iCurStationNo : INT;
	bConfirmCondition : BOOL;
	bConfirmTrigger : BOOL;
	bTransferCondition : BOOL;
	bTransferTrigger : BOOL;
	bDisable_bAvailablilityAB_Write : BOOL;

END_VAR


VAR_OUTPUT



END_VAR

VAR

	bConfirmTriggerDIFU : R_TRIG;
	TransferTriggerDIFU : R_TRIG;
	EmptyDsBasketInfo : DSV2_BasketInfo;
	iCTCompareResult: DINT;
	iTTCompareResult: DINT;
	bConfirmTriggerHR: BOOL;
	tConfirmTriggerDoff: TON;
	tTransferTriggerDoff: TON;
	bTransferTriggerHR: BOOL;
	tPreTransBasketTimer: TON;
	tCurConfirmBasketTimer: TON;
	tCurTransBasketTimer: TON;
	tPreTransBasketResetTimer: TON;
	tCurConfirmBasketResetTimer: TON;
	tCurTransBasketResetTimer: TON;
END_VAR

VAR_IN_OUT
	DSPreTransBasketInfo : DSV2_BasketInfo;
	DSCurConfirmBasketInfo : DSV2_BasketInfo;
	DSCurTransBasketInfo : DSV2_BasketInfo;

(*
	bPreTransBasket : BOOL;
	bCurConfirmBasket : BOOL;
	bCurTransBasket : BOOL;

	sPreTransStringMemory1 : STRING(50);
	sPreTransStringMemory2 : STRING(50);
	sPreTransStringMemory3 : STRING(50);
	sPreTransStringMemory4 : STRING(50);
	sPreTransStringMemory5 : STRING(50);
	sPreTransStringMemory6 : STRING(50);
	iPreTransRecipeNo : INT;
	iPrePickedBasketStationNo : INT;

	sCurConfirmStringMemory1 : STRING(50);
	sCurConfirmStringMemory2 : STRING(50);
	sCurConfirmStringMemory3 : STRING(50);
	sCurConfirmStringMemory4 : STRING(50);
	sCurConfirmStringMemory5 : STRING(50);
	sCurConfirmStringMemory6 : STRING(50);
	iCurConfirmRecipeNo : INT;



	sCurTransStringMemory1 : STRING(50);
	sCurTransStringMemory2 : STRING(50);
	sCurTransStringMemory3 : STRING(50);
	sCurTransStringMemory4 : STRING(50);
	sCurTransStringMemory5 : STRING(50);
	sCurTransStringMemory6 : STRING(50);
	iCurTransRecipeNo : INT;
	iCurPickedBasketStationNo : INT;

*)
END_VAR

(*Generate Basket Confirm Bit *)

IF DSPreTransBasketInfo.iProductRecipeNo <> 0 THEN
DSPreTransBasketInfo.bAvailibility := TRUE;
ELSE
DSPreTransBasketInfo.bAvailibility := FALSE;
END_IF

IF DSCurConfirmBasketInfo.iProductRecipeNo <> 0 THEN
DSCurConfirmBasketInfo.bAvailibility := TRUE;
ELSE
DSCurConfirmBasketInfo.bAvailibility := FALSE;
END_IF

IF DSCurTransBasketInfo.iProductRecipeNo <> 0 THEN
DSCurTransBasketInfo.bAvailibility := TRUE;
ELSE
DSCurTransBasketInfo.bAvailibility := FALSE;
END_IF

tPreTransBasketTimer(IN:= NOT bDisable_bAvailablilityAB_Write AND DSPreTransBasketInfo.bAvailibility AND NOT DSPreTransBasketInfo.bAvailibility_A AND NOT DSPreTransBasketInfo.bAvailibility_B , PT:= t#0.2s , Q=> , ET=> );
tCurConfirmBasketTimer(IN:= NOT bDisable_bAvailablilityAB_Write AND DSCurConfirmBasketInfo.bAvailibility AND NOT DSCurConfirmBasketInfo.bAvailibility_A AND NOT DSCurConfirmBasketInfo.bAvailibility_B , PT:= t#0.2s , Q=> , ET=> );
tCurTransBasketTimer(IN:= NOT bDisable_bAvailablilityAB_Write AND DSCurTransBasketInfo.bAvailibility AND NOT DSCurTransBasketInfo.bAvailibility_A AND NOT DSCurTransBasketInfo.bAvailibility_B , PT:= t#0.2s , Q=> , ET=> );

IF tPreTransBasketTimer.Q THEN
DSPreTransBasketInfo.bAvailibility_A := TRUE;
DSPreTransBasketInfo.bAvailibility_B := TRUE;
END_IF

IF tCurConfirmBasketTimer.Q THEN
DSCurConfirmBasketInfo.bAvailibility_A := TRUE;
DSCurConfirmBasketInfo.bAvailibility_B := TRUE;
END_IF

IF tCurTransBasketTimer.Q THEN
DSCurTransBasketInfo.bAvailibility_A := TRUE;
DSCurTransBasketInfo.bAvailibility_B := TRUE;
END_IF

tPreTransBasketResetTimer(IN:= NOT  DSPreTransBasketInfo.bAvailibility AND (DSPreTransBasketInfo.bAvailibility_A OR DSPreTransBasketInfo.bAvailibility_B) , PT:= t#0.1s , Q=> , ET=> );
tCurConfirmBasketResetTimer(IN:= NOT  DSCurConfirmBasketInfo.bAvailibility AND (DSCurConfirmBasketInfo.bAvailibility_A OR DSCurConfirmBasketInfo.bAvailibility_B) , PT:= t#0.1s , Q=> , ET=> );
tCurTransBasketResetTimer(IN:= NOT  DSCurTransBasketInfo.bAvailibility AND (DSCurTransBasketInfo.bAvailibility_A OR DSCurTransBasketInfo.bAvailibility_B) , PT:= t#0.1s , Q=> , ET=> );

IF tPreTransBasketResetTimer.Q THEN
DSPreTransBasketInfo.bAvailibility_A := FALSE;
DSPreTransBasketInfo.bAvailibility_B := FALSE;
END_IF

IF tCurConfirmBasketResetTimer.Q THEN
DSCurConfirmBasketInfo.bAvailibility_A := FALSE;
DSCurConfirmBasketInfo.bAvailibility_B := FALSE;
END_IF

IF tCurTransBasketResetTimer.Q THEN
DSCurTransBasketInfo.bAvailibility_A := FALSE;
DSCurTransBasketInfo.bAvailibility_B := FALSE;
END_IF








(* PreTrans -> CurConfirm *)
bConfirmTriggerDIFU(CLK:=bConfirmTrigger , Q=> );
tConfirmTriggerDoff(IN:=bConfirmTriggerHR , PT:=t#1s , Q=> , ET=> );


IF tConfirmTriggerDoff.Q THEN
bConfirmTriggerHR := FALSE;
END_IF


IF bConfirmTriggerDIFU.Q THEN
bConfirmTriggerHR := TRUE;
END_IF


IF (*bConfirmTriggerHR*)bConfirmTriggerDIFU.Q AND bConfirmCondition THEN

	IF DSPreTransBasketInfo.iProductRecipeNo <> 0 AND DSCurConfirmBasketInfo.iProductRecipeNo = 0 THEN

			DSCurConfirmBasketInfo := DSPreTransBasketInfo;

			iCTCompareResult := MEMCMP(ADR(DSCurConfirmBasketInfo), ADR(DSPreTransBasketInfo), SIZEOF(DSPreTransBasketInfo));

			IF iCTCompareResult = 0 THEN
			DSPreTransBasketInfo := EmptyDsBasketInfo;
			DSCurConfirmBasketInfo.iCurrentStationNo := iCurStationNo;
			END_IF


			IF DSCurConfirmBasketInfo.iProductRecipeNo <> 0 THEN
			DSCurConfirmBasketInfo.iPreviousStationNo := 0;
			END_IF

	END_IF

END_IF

(* CurConfirm -> CurTransfer *)
TransferTriggerDIFU(CLK:=bTransferTrigger , Q=> );

tTransferTriggerDoff(IN:=bTransferTriggerHR , PT:=t#1s , Q=> , ET=> );


IF tTransferTriggerDoff.Q THEN
bTransferTriggerHR := FALSE;
END_IF


IF TransferTriggerDIFU.Q THEN
bTransferTriggerHR := TRUE;
END_IF



IF (*bTransferTriggerHR*)TransferTriggerDIFU.Q AND bTransferCondition THEN


	IF DSCurConfirmBasketInfo.iProductRecipeNo <> 0 AND DSCurTransBasketInfo.iProductRecipeNo = 0 THEN
			DSCurTransBasketInfo := DSCurConfirmBasketInfo;

			iTTCompareResult := MEMCMP(ADR(DSCurTransBasketInfo), ADR(DSCurConfirmBasketInfo), SIZEOF(DSCurConfirmBasketInfo));

			IF iTTCompareResult = 0 THEN
			DSCurConfirmBasketInfo := EmptyDsBasketInfo;
			DSCurTransBasketInfo.iPreviousStationNo := iCurStationNo;
			END_IF


			IF DSCurTransBasketInfo.iProductRecipeNo <> 0 THEN
			DSCurTransBasketInfo.iCurrentStationNo := 0;
			END_IF

	END_IF


END_IF

END_FUNCTION_BLOCK

// ---- POUs/MainProgram/BasketMemory_RecipeCtrl/BasketToleranceCtrl.TcPOU
PROGRAM BasketToleranceCtrl
VAR
	ARfbStnToleranceCtrl		: ARRAY [0..iStnQty] OF fbToleranceTimeCtrl;

	tArm1ToleranceTimer		: TON;
	tArm1ToleranceTimerEV	: TIME;

	tArm2ToleranceTimer		: TON;
	tArm2ToleranceTimerEV	: TIME;

END_VAR

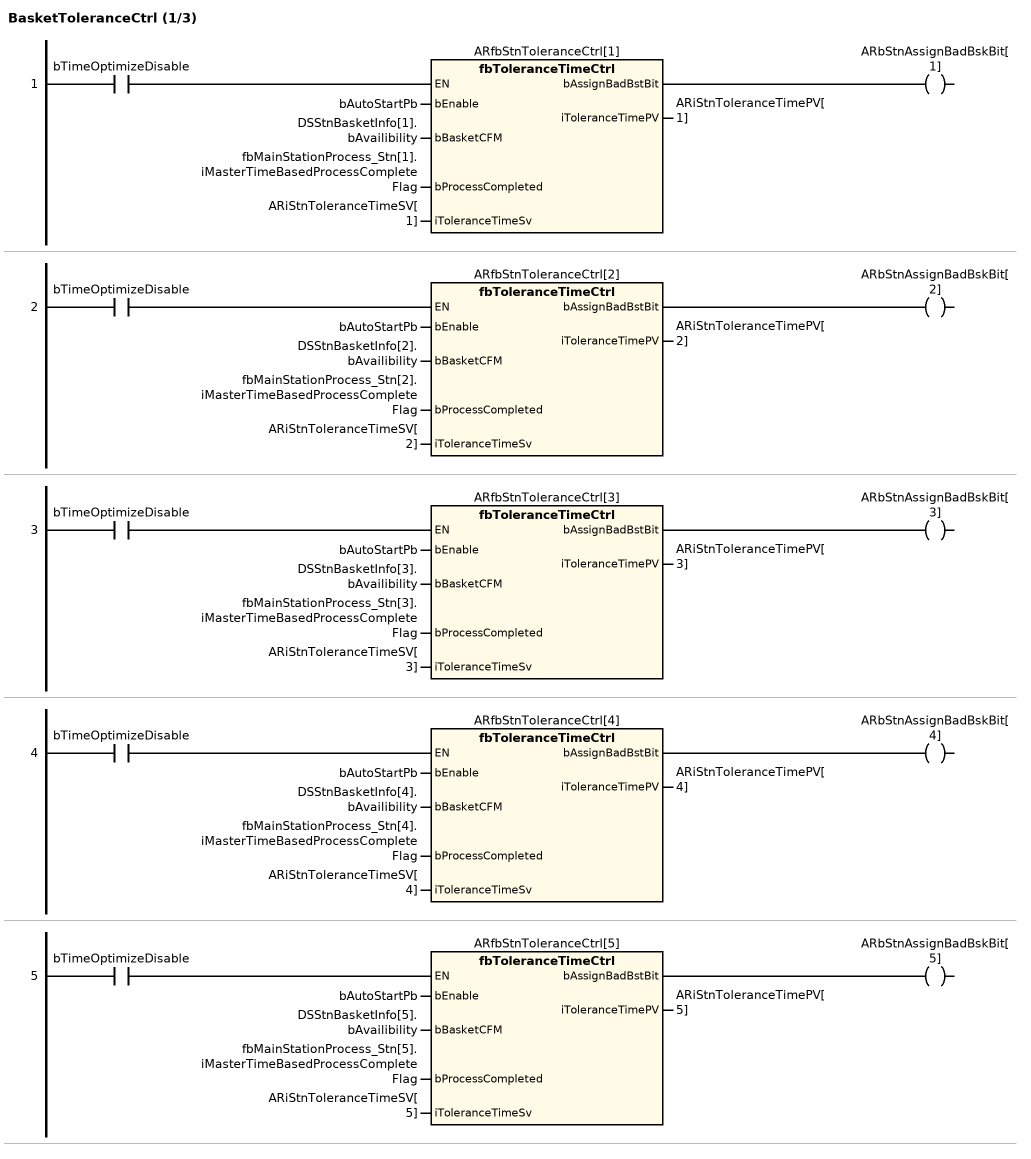
// NETWORK 1
IF bTimeOptimizeDisable THEN
    ARfbStnToleranceCtrl[1](
        bEnable := bAutoStartPb,
        bBasketCFM := DSStnBasketInfo[1].bAvailibility,
        bProcessCompleted := fbMainStationProcess_Stn[1].iMasterTimeBasedProcessCompleteFlag,
        iToleranceTimeSv := ARiStnToleranceTimeSV[1],
        iToleranceTimePV => ARiStnToleranceTimePV[1]); // fbToleranceTimeCtrl
END_IF
ARbStnAssignBadBskBit[1] := ARfbStnToleranceCtrl[1].bAssignBadBstBit;

// NETWORK 2
IF bTimeOptimizeDisable THEN
    ARfbStnToleranceCtrl[2](
        bEnable := bAutoStartPb,
        bBasketCFM := DSStnBasketInfo[2].bAvailibility,
        bProcessCompleted := fbMainStationProcess_Stn[2].iMasterTimeBasedProcessCompleteFlag,
        iToleranceTimeSv := ARiStnToleranceTimeSV[2],
        iToleranceTimePV => ARiStnToleranceTimePV[2]); // fbToleranceTimeCtrl
END_IF
ARbStnAssignBadBskBit[2] := ARfbStnToleranceCtrl[2].bAssignBadBstBit;

// NETWORK 3
IF bTimeOptimizeDisable THEN
    ARfbStnToleranceCtrl[3](
        bEnable := bAutoStartPb,
        bBasketCFM := DSStnBasketInfo[3].bAvailibility,
        bProcessCompleted := fbMainStationProcess_Stn[3].iMasterTimeBasedProcessCompleteFlag,
        iToleranceTimeSv := ARiStnToleranceTimeSV[3],
        iToleranceTimePV => ARiStnToleranceTimePV[3]); // fbToleranceTimeCtrl
END_IF
ARbStnAssignBadBskBit[3] := ARfbStnToleranceCtrl[3].bAssignBadBstBit;

// NETWORK 4
IF bTimeOptimizeDisable THEN
    ARfbStnToleranceCtrl[4](
        bEnable := bAutoStartPb,
        bBasketCFM := DSStnBasketInfo[4].bAvailibility,
        bProcessCompleted := fbMainStationProcess_Stn[4].iMasterTimeBasedProcessCompleteFlag,
        iToleranceTimeSv := ARiStnToleranceTimeSV[4],
        iToleranceTimePV => ARiStnToleranceTimePV[4]); // fbToleranceTimeCtrl
END_IF
ARbStnAssignBadBskBit[4] := ARfbStnToleranceCtrl[4].bAssignBadBstBit;

// NETWORK 5
IF bTimeOptimizeDisable THEN
    ARfbStnToleranceCtrl[5](
        bEnable := bAutoStartPb,
        bBasketCFM := DSStnBasketInfo[5].bAvailibility,
        bProcessCompleted := fbMainStationProcess_Stn[5].iMasterTimeBasedProcessCompleteFlag,
        iToleranceTimeSv := ARiStnToleranceTimeSV[5],
        iToleranceTimePV => ARiStnToleranceTimePV[5]); // fbToleranceTimeCtrl
END_IF
ARbStnAssignBadBskBit[5] := ARfbStnToleranceCtrl[5].bAssignBadBstBit;

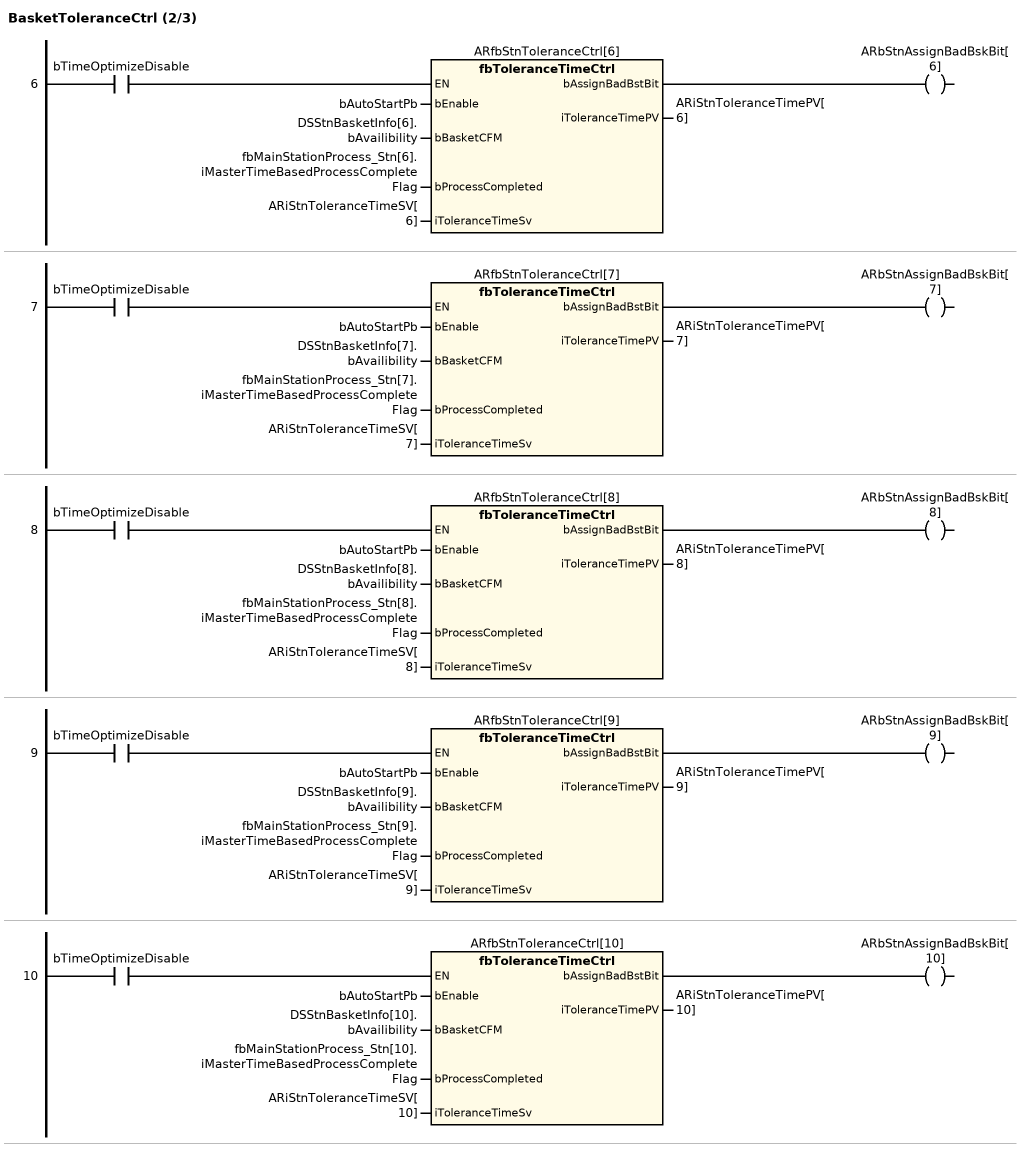
// NETWORK 6
IF bTimeOptimizeDisable THEN
    ARfbStnToleranceCtrl[6](
        bEnable := bAutoStartPb,
        bBasketCFM := DSStnBasketInfo[6].bAvailibility,
        bProcessCompleted := fbMainStationProcess_Stn[6].iMasterTimeBasedProcessCompleteFlag,
        iToleranceTimeSv := ARiStnToleranceTimeSV[6],
        iToleranceTimePV => ARiStnToleranceTimePV[6]); // fbToleranceTimeCtrl
END_IF
ARbStnAssignBadBskBit[6] := ARfbStnToleranceCtrl[6].bAssignBadBstBit;

// NETWORK 7
IF bTimeOptimizeDisable THEN
    ARfbStnToleranceCtrl[7](
        bEnable := bAutoStartPb,
        bBasketCFM := DSStnBasketInfo[7].bAvailibility,
        bProcessCompleted := fbMainStationProcess_Stn[7].iMasterTimeBasedProcessCompleteFlag,
        iToleranceTimeSv := ARiStnToleranceTimeSV[7],
        iToleranceTimePV => ARiStnToleranceTimePV[7]); // fbToleranceTimeCtrl
END_IF
ARbStnAssignBadBskBit[7] := ARfbStnToleranceCtrl[7].bAssignBadBstBit;

// NETWORK 8
IF bTimeOptimizeDisable THEN
    ARfbStnToleranceCtrl[8](
        bEnable := bAutoStartPb,
        bBasketCFM := DSStnBasketInfo[8].bAvailibility,
        bProcessCompleted := fbMainStationProcess_Stn[8].iMasterTimeBasedProcessCompleteFlag,
        iToleranceTimeSv := ARiStnToleranceTimeSV[8],
        iToleranceTimePV => ARiStnToleranceTimePV[8]); // fbToleranceTimeCtrl
END_IF
ARbStnAssignBadBskBit[8] := ARfbStnToleranceCtrl[8].bAssignBadBstBit;

// NETWORK 9
IF bTimeOptimizeDisable THEN
    ARfbStnToleranceCtrl[9](
        bEnable := bAutoStartPb,
        bBasketCFM := DSStnBasketInfo[9].bAvailibility,
        bProcessCompleted := fbMainStationProcess_Stn[9].iMasterTimeBasedProcessCompleteFlag,
        iToleranceTimeSv := ARiStnToleranceTimeSV[9],
        iToleranceTimePV => ARiStnToleranceTimePV[9]); // fbToleranceTimeCtrl
END_IF
ARbStnAssignBadBskBit[9] := ARfbStnToleranceCtrl[9].bAssignBadBstBit;

// NETWORK 10
IF bTimeOptimizeDisable THEN
    ARfbStnToleranceCtrl[10](
        bEnable := bAutoStartPb,
        bBasketCFM := DSStnBasketInfo[10].bAvailibility,
        bProcessCompleted := fbMainStationProcess_Stn[10].iMasterTimeBasedProcessCompleteFlag,
        iToleranceTimeSv := ARiStnToleranceTimeSV[10],
        iToleranceTimePV => ARiStnToleranceTimePV[10]); // fbToleranceTimeCtrl
END_IF
ARbStnAssignBadBskBit[10] := ARfbStnToleranceCtrl[10].bAssignBadBstBit;

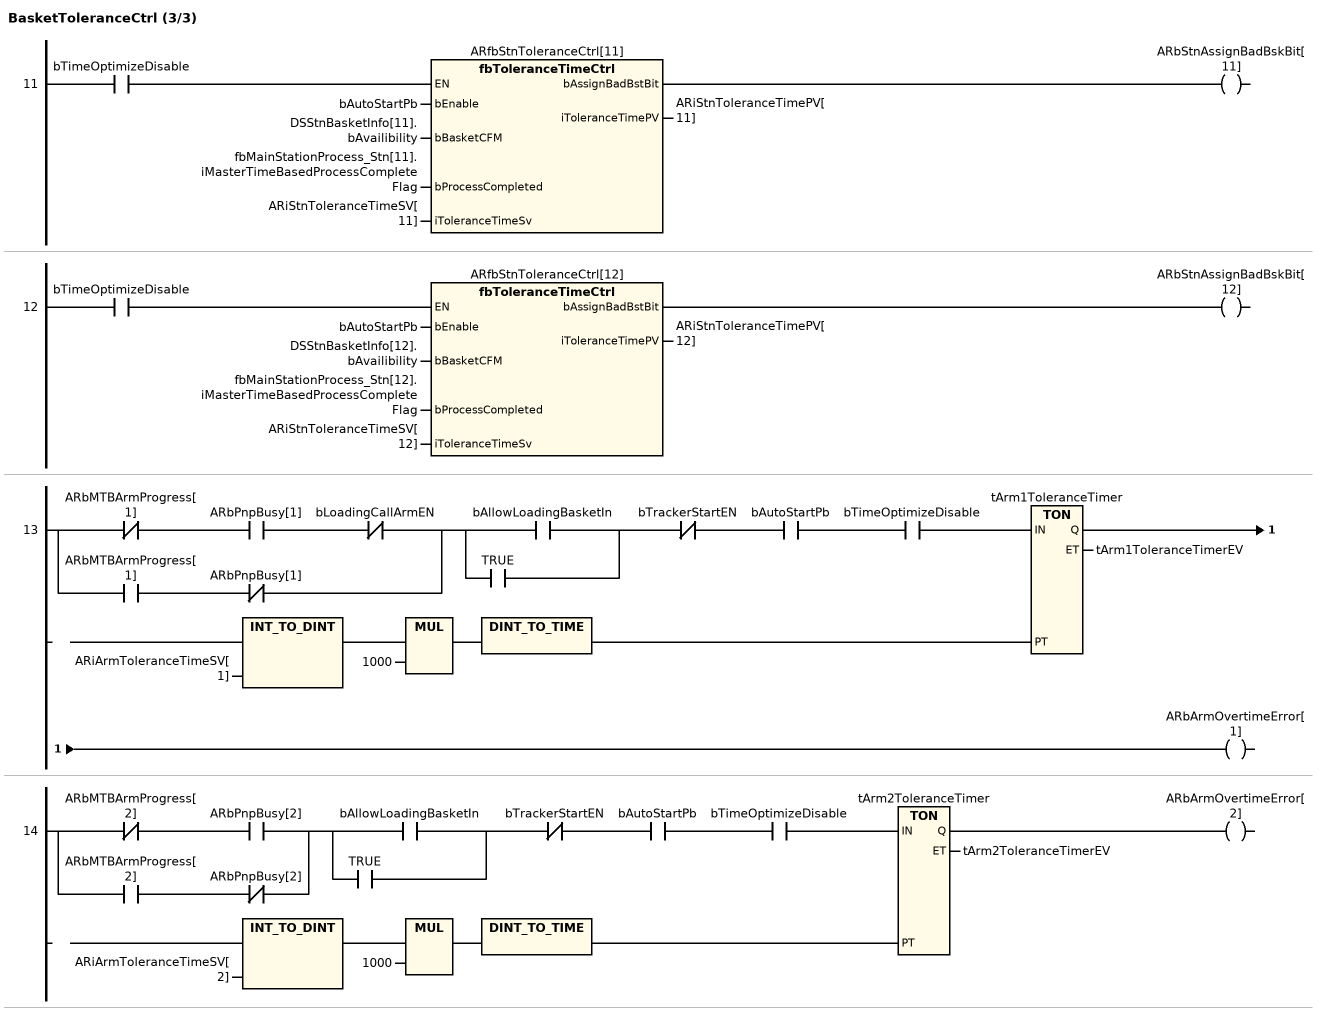
// NETWORK 11
IF bTimeOptimizeDisable THEN
    ARfbStnToleranceCtrl[11](
        bEnable := bAutoStartPb,
        bBasketCFM := DSStnBasketInfo[11].bAvailibility,
        bProcessCompleted := fbMainStationProcess_Stn[11].iMasterTimeBasedProcessCompleteFlag,
        iToleranceTimeSv := ARiStnToleranceTimeSV[11],
        iToleranceTimePV => ARiStnToleranceTimePV[11]); // fbToleranceTimeCtrl
END_IF
ARbStnAssignBadBskBit[11] := ARfbStnToleranceCtrl[11].bAssignBadBstBit;

// NETWORK 12
IF bTimeOptimizeDisable THEN
    ARfbStnToleranceCtrl[12](
        bEnable := bAutoStartPb,
        bBasketCFM := DSStnBasketInfo[12].bAvailibility,
        bProcessCompleted := fbMainStationProcess_Stn[12].iMasterTimeBasedProcessCompleteFlag,
        iToleranceTimeSv := ARiStnToleranceTimeSV[12],
        iToleranceTimePV => ARiStnToleranceTimePV[12]); // fbToleranceTimeCtrl
END_IF
ARbStnAssignBadBskBit[12] := ARfbStnToleranceCtrl[12].bAssignBadBstBit;

// NETWORK 13
tArm1ToleranceTimer(
    IN := ((NOT ARbMTBArmProgress[1] AND ARbPnpBusy[1] AND NOT bLoadingCallArmEN OR ARbMTBArmProgress[1] AND NOT ARbPnpBusy[1]) AND (bAllowLoadingBasketIn OR TRUE)) AND NOT bTrackerStartEN AND bAutoStartPb AND bTimeOptimizeDisable,
    PT := DINT_TO_TIME(INT_TO_DINT(ARiArmToleranceTimeSV[1]) * 1000),
    ET => tArm1ToleranceTimerEV); // TON
ARbArmOvertimeError[1] := tArm1ToleranceTimer.Q;

// NETWORK 14
tArm2ToleranceTimer(
    IN := ((NOT ARbMTBArmProgress[2] AND ARbPnpBusy[2] OR ARbMTBArmProgress[2] AND NOT ARbPnpBusy[2]) AND (bAllowLoadingBasketIn OR TRUE)) AND NOT bTrackerStartEN AND bAutoStartPb AND bTimeOptimizeDisable,
    PT := DINT_TO_TIME(INT_TO_DINT(ARiArmToleranceTimeSV[2]) * 1000),
    ET => tArm2ToleranceTimerEV); // TON
ARbArmOvertimeError[2] := tArm2ToleranceTimer.Q;

END_PROGRAM

// ---- FBs/B_JKS_CustomFB/fbGeneralfbFolder/fbToleranceTimeCtrl.TcPOU
FUNCTION_BLOCK fbToleranceTimeCtrl
VAR_INPUT

	bEnable					: BOOL;
	bBasketCFM				: BOOL;
	bProcessCompleted		: BOOL;
	iToleranceTimeSv		: INT;


END_VAR
VAR_OUTPUT

	bAssignBadBstBit		: BOOL;
	iToleranceTimePV	: INT;

END_VAR
VAR
	TON1: TON;
	TON2: TON;
	bAssignBadBstBitInt: BOOL;
END_VAR
VAR // added by the converter: edge detectors and wires of the graphical bodies
    _w1 : ANY;
    _w2 : INT;
END_VAR

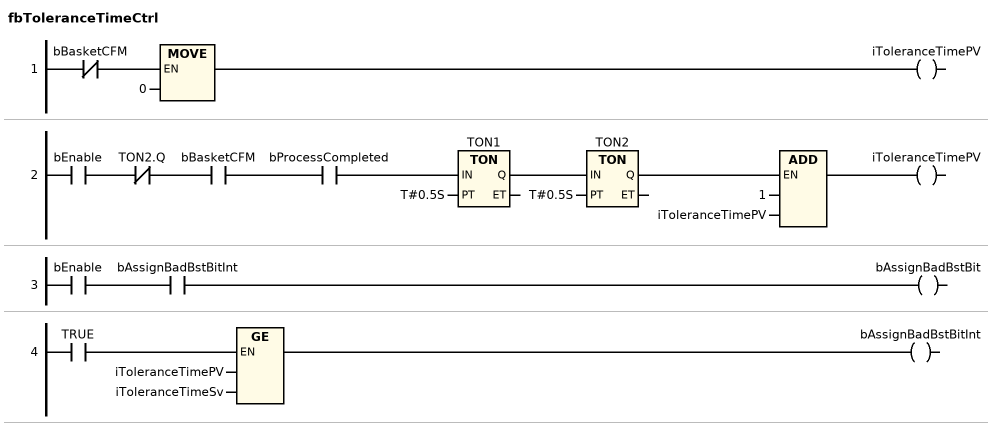
// NETWORK 1
IF NOT bBasketCFM THEN _w1 := 0; END_IF
iToleranceTimePV := _w1;

// NETWORK 2
TON1(IN := bEnable AND NOT TON2.Q AND bBasketCFM AND bProcessCompleted, PT := T#0.5S); // TON
TON2(IN := TON1.Q, PT := T#0.5S); // TON
IF TON2.Q THEN _w2 := 1 + iToleranceTimePV; END_IF
iToleranceTimePV := _w2;

// NETWORK 3
bAssignBadBstBit := bEnable AND bAssignBadBstBitInt;

// NETWORK 4
bAssignBadBstBitInt := iToleranceTimePV >= iToleranceTimeSv;

END_FUNCTION_BLOCK

// ---- POUs/MainProgram/BasketMemory_RecipeCtrl/BskMemoryCtrl.TcPOU
PROGRAM BskMemoryCtrl
VAR

	iMFL: INT;
	iSFL: INT;
	ARbLdBasketClearPb: ARRAY [1..iLdStnQty] OF BOOL;
	ARbUldBasketClearPb: ARRAY [1..iUldStnQty] OF BOOL;
	ARbLdBasketClearPbRE: R_TRIG;
	ARbUld1BasketClearPbRE: R_TRIG;
	ARbUld2BasketClearPbRE: R_TRIG;

	bCvLdBasket3ConfirmRE: R_TRIG;
	bCvLdBasket3ConfirmFE: F_TRIG;

	bCvUld1Basket1ConfirmRE: R_TRIG;
	bCvUld1Basket1ConfirmFE: F_TRIG;

	bCvUld2Basket1ConfirmRE: R_TRIG;
	bCvUld2Basket1ConfirmFE: F_TRIG;

	DSV2BasketInfoEmpty: DSV2_BasketInfo;
	ARsBarcodeDataEmpty : ARRAY [0..10] OF STRING(99); (* Byte "n+400~n+499" *)
	DSV2MinMaxEffTimeEmpty : DSV2_MinMaxEffTime;
	Nothing: BOOL;
	Nothing2: BOOL;


	(*Added for Basket Memory Control*)
(*	iLdStnQty								: INT := 1;							(* To Define Loading Group Set - How many set of Loading Conveyor*)
	iUldStnQty								: INT := 1;							(* To Define Unloading Group Set - How many set of Unloading Conveyor*)
	iCvLdQty									: INT := 1;
	iCvUldQty								: INT := 1;
	iStnQty 									: INT := 10;						(* To change the Qty of Array*)
	iArmQty 									: INT := 1; 						(* ArmQty must lesser than StnQty*)
*)
(*
	fbBasketInfoManagerCfm_STN : ARRAY [0..iStnQty] OF fbV2_BasketInfoManager;

	fbBasketInfoManagerCfm_ARM : ARRAY [0..iArmQty] OF fbV2_BasketInfoManager;


	DSLdBasketInfoConfirm 				: ARRAY [0..iLdStnQty] OF DSV2_BasketInfo;
	DSLdBasketInfoTransfer 				: ARRAY [0..iLdStnQty] OF DSV2_BasketInfo;

	DSUldBasketInfoConfirm 				: ARRAY [0..iUldStnQty] OF DSV2_BasketInfo;
	DSUldBasketInfoTransfer 				: ARRAY [0..iUldStnQty] OF DSV2_BasketInfo;

	DSStnBasketInfo						: ARRAY [0..iStnQty] OF DSV2_BasketInfo;
	DSArmBasketInfo 						: ARRAY [0..iArmQty] OF DSV2_BasketInfo;

*)

	iBMFL: INT;
	iBMSFL: INT;
END_VAR

(*xxxxxxxxxxxxxxxxxxxxxxxxx Basket Memory Clear - Loading / Unloading Control xxxxxxxxxxxxxxxxxxxxxxxxx*)
ARbLdBasketClearPbRE(CLK:= ARbLdBasketClearPb[1] , Q=> );
ARbUld1BasketClearPbRE(CLK:= ARbUldBasketClearPb[1] , Q=> );
(*ARbUld2BasketClearPbRE(CLK:= ARbUldBasketClearPb[2] , Q=> );*)

IF ARbLdBasketClearPbRE.Q THEN
		iSFL :=1;
			FOR iSFL := 1 TO iCvLdQty DO
				IF iSFL >= 1 AND iSFL <= iCvLdQty THEN
					AR2sDSCv_LdConfirmBasketInfo[1, iSFL].iProductRecipeNo := 0;
					AR2sDSCv_LdTransferBasketInfo[1,iSFL].iProductRecipeNo := 0;
				END_IF
			END_FOR
END_IF

IF ARbUld1BasketClearPbRE.Q THEN
		iSFL :=1;
			FOR iSFL := 1 TO iCvUldQty DO
				IF iSFL >= 1 AND iSFL <= iCvUldQty THEN
					AR2sDSCv_UldConfirmBasketInfo[1, iSFL].iProductRecipeNo := 0;
					AR2sDSCv_UldTransferBasketInfo[1,iSFL].iProductRecipeNo := 0;
				END_IF
			END_FOR
END_IF


(*
IF ARbUld2BasketClearPbRE.Q THEN
		iSFL :=1;
			FOR iSFL := 1 TO iCvUldQty DO
				IF iSFL >= 1 AND iSFL <= iCvUldQty THEN
					AR2sDSCv_UldConfirmBasketInfo[2, iSFL].iProductRecipeNo := 0;
					AR2sDSCv_UldTransferBasketInfo[2,iSFL].iProductRecipeNo := 0;
				END_IF
			END_FOR
END_IF
*)

(*xxxxxxxxxxxxxxxxxxxxxxxxx Basket Memory  - Loading Conveyor "AR2sDSCv_LdConfirmBasketInfo" MOVE to " DSLdBasketInfoConfirm Control"xxxxxxxxxxxxxxxxxxxxxxxxx*)

bCvLdBasket3ConfirmRE(CLK:=AR2sDSCv_LdConfirmBasketInfo[1,4].bAvailibility , Q=> );
IF bCvLdBasket3ConfirmRE.Q OR fbBasketInfoManagerCfm_LDCV[1,4].bRecipeChangedFlag OR fbBasketInfoManagerCfm_LDCV[1,4].bMinMaxEffChangeFlag THEN
DSLdBasketInfoConfirm[1] := AR2sDSCv_LdConfirmBasketInfo[1,4];
END_IF

bCvLdBasket3ConfirmFE(CLK:=AR2sDSCv_LdConfirmBasketInfo[1,4].bAvailibility , Q=> );
IF bCvLdBasket3ConfirmFE.Q THEN
DSLdBasketInfoConfirm[1] := DSV2BasketInfoEmpty;
END_IF

(*xxxxxxxxxxxxxxxxxxxxxxxxx Basket Memory  - Unloading Conveyor "AR2sDSCv_UldConfirmBasketInfo" MOVE to " DSUldBasketInfoConfirm Control"xxxxxxxxxxxxxxxxxxxxxxxxx*)

bCvUld1Basket1ConfirmRE(CLK:=AR2sDSCv_UldConfirmBasketInfo[1,1].bAvailibility , Q=> );
IF bCvUld1Basket1ConfirmRE.Q THEN
DSUldBasketInfoConfirm[1] := AR2sDSCv_UldConfirmBasketInfo[1,1];
END_IF


bCvUld1Basket1ConfirmFE(CLK:=AR2sDSCv_UldConfirmBasketInfo[1,1].bAvailibility , Q=> );
IF bCvUld1Basket1ConfirmFE.Q THEN
DSUldBasketInfoConfirm[1] := DSV2BasketInfoEmpty;
END_IF


(*xxxxxxxxxxxxxxxxxxxxxxxxx Basket Memory  - Loading - Station - Unloading Control xxxxxxxxxxxxxxxxxxxxxxxxx*)


iBMFL := 1;
FOR iBMFL := 1 TO iLdStnQty DO
	IF iBMFL >= 1 AND iBMFL <= iLdStnQty THEN
		iBMSFL := 1;
		FOR iBMSFL := 1 TO iCvLdQty DO
			IF iBMSFL >= 1 AND iBMSFL <= iCvLdQty THEN
				fbBasketInfoManagerCfm_LDCV[iBMFL,iBMSFL](iRecipeChangeFlagDelayTime_Sec:=0.3 , DSV2BasketInfo:=AR2sDSCv_LdConfirmBasketInfo[iBMFL,iBMSFL] , bRecipeChangedFlag=> );
				fbBasketInfoManagerTrf_LDCV[iBMFL,iBMSFL](iRecipeChangeFlagDelayTime_Sec:=0.3 , DSV2BasketInfo:=AR2sDSCv_LdTransferBasketInfo[iBMFL,iBMSFL] , bRecipeChangedFlag=> );
			END_IF
		END_FOR
	END_IF
END_FOR

iBMFL := 1;
FOR iBMFL := 1 TO iUldStnQty DO
	IF iBMFL >= 1 AND iBMFL <= iUldStnQty THEN
		iBMSFL := 1;
		FOR iBMSFL := 1 TO iCvUldQty DO
			IF iBMSFL >= 1 AND iBMSFL <= iCvUldQty THEN
				fbBasketInfoManagerCfm_ULDCV[iBMFL,iBMSFL](iRecipeChangeFlagDelayTime_Sec:=0.3 , DSV2BasketInfo:=AR2sDSCv_UldConfirmBasketInfo[iBMFL,iBMSFL] , bRecipeChangedFlag=> );
				fbBasketInfoManagerTrf_ULDCV[iBMFL,iBMSFL](iRecipeChangeFlagDelayTime_Sec:=0.3 , DSV2BasketInfo:=AR2sDSCv_UldTransferBasketInfo[iBMFL,iBMSFL] , bRecipeChangedFlag=> );
			END_IF
		END_FOR
	END_IF
END_FOR

iBMFL := 1;
FOR iBMFL := 1 TO iLdStnQty DO
	IF iBMFL >= 1 AND iBMFL <= iLdStnQty THEN
		fbBasketInfoManagerCfm_LD[iBMFL](iRecipeChangeFlagDelayTime_Sec:=0.3 , DSV2BasketInfo:=DSLdBasketInfoConfirm[iBMFL] , bRecipeChangedFlag=> );
		fbBasketInfoManagerTrf_LD[iBMFL](iRecipeChangeFlagDelayTime_Sec:=0.3 , DSV2BasketInfo:=DSLdBasketInfoTransfer[iBMFL] , bRecipeChangedFlag=> );
	END_IF
END_FOR

iBMFL := 1;
FOR iBMFL := 1 TO iUldStnQty DO
	IF iBMFL >= 1 AND iBMFL <= iUldStnQty THEN
		fbBasketInfoManagerCfm_ULD[iBMFL](iRecipeChangeFlagDelayTime_Sec:=0.3 , DSV2BasketInfo:=DSUldBasketInfoConfirm[iBMFL] , bRecipeChangedFlag=> );
		fbBasketInfoManagerTrf_ULD[iBMFL](iRecipeChangeFlagDelayTime_Sec:=0.3 , DSV2BasketInfo:=DSUldBasketInfoTransfer[iBMFL] , bRecipeChangedFlag=> );
	END_IF
END_FOR


iBMFL := 1;
FOR iBMFL := 1 TO iStnQty DO
	IF iBMFL >= 1 AND iBMFL <= iStnQty THEN
		fbBasketInfoManagerCfm_STN[iBMFL](iRecipeChangeFlagDelayTime_Sec:=0.3 , DSV2BasketInfo:=DSStnBasketInfo[iBMFL] , bRecipeChangedFlag=> );
	END_IF
END_FOR

iBMFL := 1;
FOR iBMFL := 1 TO iArmQty DO
	IF iBMFL >= 1 AND iBMFL <= iArmQty THEN
		fbBasketInfoManagerCfm_ARM[iBMFL](iRecipeChangeFlagDelayTime_Sec:=0.3 , DSV2BasketInfo:=DSArmBasketInfo[iBMFL] , bRecipeChangedFlag=> );
	END_IF
END_FOR


IF AR2sDSCv_LdConfirmBasketInfo[1,4].bAvailibility AND AR2sDSCv_LdConfirmBasketInfo[1,4].sProductQuality ='GOOD' THEN
ARbBasketGdFlag[1] := TRUE;
ELSE
ARbBasketGdFlag[1] := FALSE;
END_IF


IF DSStnBasketInfo[1].bAvailibility AND DSStnBasketInfo[1].sProductQuality ='GOOD' THEN
ARbBasketGdFlag[2] := TRUE;
ELSE
ARbBasketGdFlag[2] := FALSE;
END_IF

IF DSStnBasketInfo[2].bAvailibility AND DSStnBasketInfo[2].sProductQuality ='GOOD' THEN
ARbBasketGdFlag[3] := TRUE;
ELSE
ARbBasketGdFlag[3] := FALSE;
END_IF

IF DSStnBasketInfo[3].bAvailibility AND DSStnBasketInfo[3].sProductQuality ='GOOD' THEN
ARbBasketGdFlag[4] := TRUE;
ELSE
ARbBasketGdFlag[4] := FALSE;
END_IF

IF DSStnBasketInfo[4].bAvailibility AND DSStnBasketInfo[4].sProductQuality ='GOOD' THEN
ARbBasketGdFlag[5] := TRUE;
ELSE
ARbBasketGdFlag[5] := FALSE;
END_IF

IF DSStnBasketInfo[5].bAvailibility AND DSStnBasketInfo[5].sProductQuality ='GOOD' THEN
ARbBasketGdFlag[6] := TRUE;
ELSE
ARbBasketGdFlag[6] := FALSE;
END_IF

IF DSStnBasketInfo[6].bAvailibility AND DSStnBasketInfo[6].sProductQuality ='GOOD' THEN
ARbBasketGdFlag[7] := TRUE;
ELSE
ARbBasketGdFlag[7] := FALSE;
END_IF

IF DSStnBasketInfo[7].bAvailibility AND DSStnBasketInfo[7].sProductQuality ='GOOD' THEN
ARbBasketGdFlag[8] := TRUE;
ELSE
ARbBasketGdFlag[8] := FALSE;
END_IF

IF DSStnBasketInfo[8].bAvailibility AND DSStnBasketInfo[8].sProductQuality ='GOOD' THEN
ARbBasketGdFlag[9] := TRUE;
ELSE
ARbBasketGdFlag[9] := FALSE;
END_IF

IF DSStnBasketInfo[9].bAvailibility AND DSStnBasketInfo[9].sProductQuality ='GOOD' THEN
ARbBasketGdFlag[10] := TRUE;
ELSE
ARbBasketGdFlag[10] := FALSE;
END_IF

IF DSStnBasketInfo[10].bAvailibility AND DSStnBasketInfo[10].sProductQuality ='GOOD' THEN
ARbBasketGdFlag[11] := TRUE;
ELSE
ARbBasketGdFlag[11] := FALSE;
END_IF

IF AR2sDSCv_UldConfirmBasketInfo[1,1].bAvailibility AND AR2sDSCv_UldConfirmBasketInfo[1,1].sProductQuality ='GOOD' THEN
ARbBasketGdFlag[12] := TRUE;
ELSE
ARbBasketGdFlag[12] := FALSE;
END_IF

IF AR2sDSCv_UldConfirmBasketInfo[1,2].bAvailibility AND AR2sDSCv_UldConfirmBasketInfo[1,2].sProductQuality ='GOOD' THEN
ARbBasketGdFlag[13] := TRUE;
ELSE
ARbBasketGdFlag[13] := FALSE;
END_IF

IF AR2sDSCv_UldConfirmBasketInfo[1,3].bAvailibility AND AR2sDSCv_UldConfirmBasketInfo[1,3].sProductQuality ='GOOD' THEN
ARbBasketGdFlag[14] := TRUE;
ELSE
ARbBasketGdFlag[14] := FALSE;
END_IF

IF AR2sDSCv_UldConfirmBasketInfo[1,4].bAvailibility AND AR2sDSCv_UldConfirmBasketInfo[1,4].sProductQuality ='GOOD' THEN
ARbBasketGdFlag[15] := TRUE;
ELSE
ARbBasketGdFlag[15] := FALSE;
END_IF
(*
IF AR2sDSCv_UldConfirmBasketInfo[1,5].bAvailibility AND AR2sDSCv_UldConfirmBasketInfo[1,5].sProductQuality ='GOOD' THEN
ARbBasketGdFlag[16] := TRUE;
ELSE
ARbBasketGdFlag[16] := FALSE;
END_IF
*)

IF DSArmBasketInfo[1].bAvailibility AND DSArmBasketInfo[1].sProductQuality ='GOOD' THEN
ARbBasketGdFlag[16] := TRUE;
ELSE
ARbBasketGdFlag[16] := FALSE;
END_IF

(*
IF DSArmBasketInfo[2].bAvailibility AND DSArmBasketInfo[2].sProductQuality ='GOOD' THEN
ARbBasketGdFlag[18] := TRUE;
ELSE
ARbBasketGdFlag[18] := FALSE;
END_IF
*)


IF DSStnBasketInfo[1].bAvailibility AND DSStnBasketInfo[1].sProductQuality ='BAD' THEN
ARbBasketBdFlag[2] := TRUE;
ELSE
ARbBasketBdFlag[2] := FALSE;
END_IF

IF DSStnBasketInfo[2].bAvailibility AND DSStnBasketInfo[2].sProductQuality ='BAD' THEN
ARbBasketBdFlag[3] := TRUE;
ELSE
ARbBasketBdFlag[3] := FALSE;
END_IF

IF DSStnBasketInfo[3].bAvailibility AND DSStnBasketInfo[3].sProductQuality ='BAD' THEN
ARbBasketBdFlag[4] := TRUE;
ELSE
ARbBasketBdFlag[4] := FALSE;
END_IF

IF DSStnBasketInfo[4].bAvailibility AND DSStnBasketInfo[4].sProductQuality ='BAD' THEN
ARbBasketBdFlag[5] := TRUE;
ELSE
ARbBasketBdFlag[5] := FALSE;
END_IF

IF DSStnBasketInfo[5].bAvailibility AND DSStnBasketInfo[5].sProductQuality ='BAD' THEN
ARbBasketBdFlag[6] := TRUE;
ELSE
ARbBasketBdFlag[6] := FALSE;
END_IF

IF DSStnBasketInfo[6].bAvailibility AND DSStnBasketInfo[6].sProductQuality ='BAD' THEN
ARbBasketBdFlag[7] := TRUE;
ELSE
ARbBasketBdFlag[7] := FALSE;
END_IF

IF DSStnBasketInfo[7].bAvailibility AND DSStnBasketInfo[7].sProductQuality ='BAD' THEN
ARbBasketBdFlag[8] := TRUE;
ELSE
ARbBasketBdFlag[8] := FALSE;
END_IF

IF DSStnBasketInfo[8].bAvailibility AND DSStnBasketInfo[8].sProductQuality ='BAD' THEN
ARbBasketBdFlag[9] := TRUE;
ELSE
ARbBasketBdFlag[9] := FALSE;
END_IF

IF DSStnBasketInfo[9].bAvailibility AND DSStnBasketInfo[9].sProductQuality ='BAD' THEN
ARbBasketBdFlag[10] := TRUE;
ELSE
ARbBasketBdFlag[10] := FALSE;
END_IF

IF DSStnBasketInfo[10].bAvailibility AND DSStnBasketInfo[10].sProductQuality ='BAD' THEN
ARbBasketBdFlag[11] := TRUE;
ELSE
ARbBasketBdFlag[11] := FALSE;
END_IF
(*
IF DSStnBasketInfo[11].bAvailibility AND DSStnBasketInfo[11].sProductQuality ='BAD' THEN
ARbBasketBdFlag[12] := TRUE;
ELSE
ARbBasketBdFlag[12] := FALSE;
END_IF

IF DSStnBasketInfo[12].bAvailibility AND DSStnBasketInfo[12].sProductQuality ='BAD' THEN
ARbBasketBdFlag[13] := TRUE;
ELSE
ARbBasketBdFlag[13] := FALSE;
END_IF
*)

IF AR2sDSCv_UldConfirmBasketInfo[1,1].bAvailibility AND AR2sDSCv_UldConfirmBasketInfo[1,1].sProductQuality ='BAD' THEN
ARbBasketBdFlag[12] := TRUE;
ELSE
ARbBasketBdFlag[12] := FALSE;
END_IF

IF AR2sDSCv_UldConfirmBasketInfo[1,2].bAvailibility AND AR2sDSCv_UldConfirmBasketInfo[1,2].sProductQuality ='BAD' THEN
ARbBasketBdFlag[13] := TRUE;
ELSE
ARbBasketBdFlag[13] := FALSE;
END_IF

IF AR2sDSCv_UldConfirmBasketInfo[1,3].bAvailibility AND AR2sDSCv_UldConfirmBasketInfo[1,3].sProductQuality ='BAD' THEN
ARbBasketBdFlag[14] := TRUE;
ELSE
ARbBasketBdFlag[14] := FALSE;
END_IF

IF AR2sDSCv_UldConfirmBasketInfo[1,4].bAvailibility AND AR2sDSCv_UldConfirmBasketInfo[1,4].sProductQuality ='BAD' THEN
ARbBasketBdFlag[15] := TRUE;
ELSE
ARbBasketBdFlag[15] := FALSE;
END_IF

IF DSArmBasketInfo[1].bAvailibility AND DSArmBasketInfo[1].sProductQuality ='BAD' THEN
ARbBasketBdFlag[16] := TRUE;
ELSE
ARbBasketBdFlag[16] := FALSE;
END_IF

END_PROGRAM

// ---- POUs/MainProgram/BasketMemory_RecipeCtrl/CvMotorREFE.TcPOU
PROGRAM CvMotorREFE
VAR
END_VAR

;
(*Loading Conveyor Motor REFE*)

LdMotor1RE(CLK:= ARbDO[eY10301_LoadingConveyor01On_Off] AND ARbDO[eY10302_LoadingConveyor02On_Off] , Q=> );
LdMotor2RE(CLK:= ARbDO[eY10302_LoadingConveyor02On_Off] AND ARbDO[eY10303_LoadingConveyor03On_Off] , Q=> );
LdMotor3RE(CLK:= ARbDO[eY10303_LoadingConveyor03On_Off] AND ARbDO[eY10304_LoadingConveyor04On_Off], Q=> );
LdMotor4RE(CLK:= ARbDO[eY10304_LoadingConveyor04On_Off]  , Q=> );
(*LdMotor5RE(CLK:= Y102_01 , Q=> );*)

LdMotor1FE(CLK:= ARbDO[eY10301_LoadingConveyor01On_Off] AND ARbDO[eY10302_LoadingConveyor02On_Off], Q=> );
LdMotor2FE(CLK:= ARbDO[eY10302_LoadingConveyor02On_Off] AND ARbDO[eY10303_LoadingConveyor03On_Off], Q=> );
LdMotor3FE(CLK:= ARbDO[eY10303_LoadingConveyor03On_Off] AND ARbDO[eY10304_LoadingConveyor04On_Off] , Q=> );
LdMotor4FE(CLK:= ARbDO[eY10304_LoadingConveyor04On_Off], Q=> );
(*LdMotor5FE(CLK:= Y102_01 , Q=> );
*)

(*Unloading Conveyor Motor REFE*)

UldMotor1RE(CLK:=ARbDO[eY10305_UnloadingConveyor01On_Off] AND ARbDO[eY10306_UnloadingConveyor02On_Off], Q=> );
UldMotor2RE(CLK:=ARbDO[eY10306_UnloadingConveyor02On_Off] AND ARbDO[eY10307_UnloadingConveyor03On_Off], Q=> );
UldMotor3RE(CLK:=ARbDO[eY10307_UnloadingConveyor03On_Off] AND ARbDO[eY10308_UnloadingConveyor04On_Off], Q=> );
UldMotor4RE(CLK:=ARbDO[eY10308_UnloadingConveyor04On_Off], Q=> );
(*UldMotor5RE(CLK:= Y102_06, Q=> );
*)
UldMotor1FE(CLK:= ARbDO[eY10305_UnloadingConveyor01On_Off] AND ARbDO[eY10306_UnloadingConveyor02On_Off] , Q=> );
UldMotor2FE(CLK:= ARbDO[eY10306_UnloadingConveyor02On_Off] AND ARbDO[eY10307_UnloadingConveyor03On_Off], Q=> );
UldMotor3FE(CLK:= ARbDO[eY10307_UnloadingConveyor03On_Off] AND ARbDO[eY10308_UnloadingConveyor04On_Off], Q=> );
UldMotor4FE(CLK:= ARbDO[eY10308_UnloadingConveyor04On_Off], Q=> );

(*UldMotor5FE(CLK:= Y102_06, Q=> );

X155_00; (*FEED*)
X155_01; (*INDEX 1*) Y102_03; Y102_04;
X155_02; (*INDEX 2*) Y102_04; Y102_05;
X155_03; (*INDEX 3*) Y102_05; Y102_06;
X155_04; (*PICK*)

IF (Y101_13 OR Y101_14 OR Y101_15 OR Y102_00 OR Y102_01) THEN
bLoadingConveyorBusyFlag := TRUE;
ELSE
bLoadingConveyorBusyFlag := FALSE;
END_IF


IF (Y102_02 OR Y102_03 OR Y102_04 OR Y102_05 OR Y102_06) THEN
bUnloadingConveyorBusyFlag := TRUE;
ELSE
bUnloadingConveyorBusyFlag := FALSE;
END_IF
*)

END_PROGRAM

// ---- POUs/MainProgram/DataManagement/ArmPickTransferCtrl_General.TcPOU
PROGRAM ArmPickTransferCtrl_General
VAR
	fbGenerateArmPickTransferBit_Arm1Horz		: fbV2_GenerateArmPickTransferBit;

END_VAR

